LIN {X 0,Y 580.158,Z 386.279,A -85,B 0,C 180,E1 -1986.958,E2 -1986.958} C_VEL
LIN {X 0,Y 580.242,Z 378.359,A -85,B 0,C 180,E1 -1988.007,E2 -1988.007} C_VEL
LIN {X 0,Y 580.308,Z 368.509,A -85,B 0,C 180,E1 -1989.058,E2 -1989.058} C_VEL
LIN {X 0,Y 580.415,Z 358.188,A -85,B 0,C 180,E1 -1989.936,E2 -1989.936} C_VEL
LIN {X 0,Y 580.533,Z 346.552,A -85,B 0,C 180,E1 -1990.727,E2 -1990.727} C_VEL
LIN {X 0,Y 580.614,Z 334.997,A -85,B 0,C 180,E1 -1991.344,E2 -1991.344} C_VEL
LIN {X 0,Y 580.632,Z 322.991,A -85,B 0,C 180,E1 -1991.83,E2 -1991.83} C_VEL
LIN {X 0,Y 580.756,Z 309.958,A -85,B 0,C 180,E1 -1992.204,E2 -1992.204} C_VEL
LIN {X 0,Y 580.802,Z 297.624,A -85,B 0,C 180,E1 -1992.425,E2 -1992.425} C_VEL
LIN {X 0,Y 580.926,Z 253.863,A -85,B 0,C 180,E1 -1992.966,E2 -1992.966} C_VEL
LIN {X 0,Y 580.276,Z 248.059,A -85,B 0,C 180,E1 -1993.053,E2 -1993.053} C_VEL
LIN {X 0,Y 574.724,Z 229.373,A -85,B 0,C 180,E1 -1993.416,E2 -1993.416} C_VEL
LIN {X 0,Y 574.032,Z 223.57,A -85,B 0,C 180,E1 -1993.505,E2 -1993.505} C_VEL
LIN {X 0,Y 573.952,Z 199.2,A -85,B 0,C 180,E1 -1993.814,E2 -1993.814} C_VEL
LIN {X 0,Y 573.397,Z 195.222,A -85,B 0,C 180,E1 -1993.896,E2 -1993.896} C_VEL
LIN {X 0,Y 573.541,Z 175.453,A -85,B 0,C 180,E1 -1996.722,E2 -1996.722} C_VEL
LIN {X 0,Y 573.812,Z 157.024,A -85,B 0,C 180,E1 -1999.422,E2 -1999.422} C_VEL
LIN {X 0,Y 574.091,Z 137.477,A -85,B 0,C 180,E1 -2002.303,E2 -2002.303} C_VEL
LIN {X 0,Y 573.843,Z 133.661,A -85,B 0,C 180,E1 -2002.883,E2 -2002.883} C_VEL
LIN {X 0,Y 573.232,Z 130.71,A -85,B 0,C 180,E1 -2003.377,E2 -2003.377} C_VEL
LIN {X 0,Y 573.247,Z 130.708,A -85,B 0,C 180,E1 -2005.411,E2 -2005.411} C_VEL
LIN {X 0,Y 573.226,Z 130.702,A -85,B 0,C 180,E1 -2008.565,E2 -2008.565} C_VEL
LIN {X 0,Y 573.222,Z 130.705,A -85,B 0,C 180,E1 -2010.994,E2 -2010.994} C_VEL
LIN {X 0,Y 573.268,Z 130.704,A -85,B 0,C 180,E1 -2013.524,E2 -2013.524} C_VEL
LIN {X 0,Y 573.197,Z 130.706,A -85,B 0,C 180,E1 -2016.053,E2 -2016.053} C_VEL
LIN {X 0,Y 573.242,Z 130.701,A -85,B 0,C 180,E1 -2018.702,E2 -2018.702} C_VEL
LIN {X 0,Y 573.218,Z 130.706,A -85,B 0,C 180,E1 -2021.591,E2 -2021.591} C_VEL
LIN {X 0,Y 573.229,Z 130.7,A -85,B 0,C 180,E1 -2024.334,E2 -2024.334} C_VEL
LIN {X 0,Y 573.242,Z 130.704,A -85,B 0,C 180,E1 -2027.358,E2 -2027.358} C_VEL
LIN {X 0,Y 573.241,Z 130.701,A -85,B 0,C 180,E1 -2030.392,E2 -2030.392} C_VEL
LIN {X 0,Y 573.256,Z 130.705,A -85,B 0,C 180,E1 -2033.077,E2 -2033.077} C_VEL
LIN {X 0,Y 573.26,Z 130.698,A -85,B 0,C 180,E1 -2035.67,E2 -2035.67} C_VEL
LIN {X 0,Y 573.243,Z 130.702,A -85,B 0,C 180,E1 -2038.184,E2 -2038.184} C_VEL
LIN {X 0,Y 573.263,Z 130.706,A -85,B 0,C 180,E1 -2040.633,E2 -2040.633} C_VEL
LIN {X 0,Y 573.239,Z 130.701,A -85,B 0,C 180,E1 -2043.507,E2 -2043.507} C_VEL
LIN {X 0,Y 573.231,Z 130.708,A -85,B 0,C 180,E1 -2046.134,E2 -2046.134} C_VEL
LIN {X 0,Y 573.288,Z 130.867,A -85,B 0,C 180,E1 -2046.773,E2 -2046.773} C_VEL
LIN {X 0,Y 574.099,Z 135.892,A -85,B 0,C 180,E1 -2047.507,E2 -2047.507} C_VEL
LIN {X 0,Y 573.843,Z 156.505,A -85,B 0,C 180,E1 -2050.382,E2 -2050.382} C_VEL
LIN {X 0,Y 573.897,Z 157.389,A -85,B 0,C 180,E1 -2050.451,E2 -2050.451} C_VEL
LIN {X 0,Y 575.176,Z 163.348,A -85,B 0,C 180,E1 -2050.573,E2 -2050.573} C_VEL
LIN {X 0,Y 574.754,Z 320.455,A -85,B 0,C 180,E1 -2052.605,E2 -2052.605} C_VEL
LIN {X 0,Y 574.634,Z 333.869,A -85,B 0,C 180,E1 -2052.88,E2 -2052.88} C_VEL
LIN {X 0,Y 574.472,Z 349.297,A -85,B 0,C 180,E1 -2053.337,E2 -2053.337} C_VEL
LIN {X 0,Y 574.303,Z 363.777,A -85,B 0,C 180,E1 -2053.926,E2 -2053.926} C_VEL
LIN {X 0,Y 574.121,Z 376.223,A -85,B 0,C 180,E1 -2054.558,E2 -2054.558} C_VEL
LIN {X 0,Y 573.959,Z 387.161,A -85,B 0,C 180,E1 -2055.222,E2 -2055.222} C_VEL
LIN {X 0,Y 573.735,Z 398.068,A -85,B 0,C 180,E1 -2055.999,E2 -2055.999} C_VEL
LIN {X 0,Y 573.576,Z 408.837,A -85,B 0,C 180,E1 -2056.898,E2 -2056.898} C_VEL
LIN {X 0,Y 573.4,Z 421.37,A -85,B 0,C 180,E1 -2058.152,E2 -2058.152} C_VEL
LIN {X 0,Y 573.312,Z 430.525,A -85,B 0,C 180,E1 -2059.257,E2 -2059.257} C_VEL
LIN {X 0,Y 573.195,Z 437.937,A -85,B 0,C 180,E1 -2060.293,E2 -2060.293} C_VEL
LIN {X 0,Y 573.113,Z 445.456,A -85,B 0,C 180,E1 -2061.537,E2 -2061.537} C_VEL
LIN {X 0,Y 573.05,Z 452.505,A -85,B 0,C 180,E1 -2062.955,E2 -2062.955} C_VEL
LIN {X 0,Y 573.055,Z 458.02,A -85,B 0,C 180,E1 -2064.369,E2 -2064.369} C_VEL
LIN {X 0,Y 573.008,Z 462.158,A -85,B 0,C 180,E1 -2065.779,E2 -2065.779} C_VEL
LIN {X 0,Y 572.954,Z 465.104,A -85,B 0,C 180,E1 -2067.187,E2 -2067.187} C_VEL
LIN {X 0,Y 572.943,Z 466.876,A -85,B 0,C 180,E1 -2068.593,E2 -2068.593} C_VEL
LIN {X 0,Y 572.936,Z 467.496,A -85,B 0,C 180,E1 -2069.999,E2 -2069.999} C_VEL
LIN {X 0,Y 572.945,Z 466.961,A -85,B 0,C 180,E1 -2071.405,E2 -2071.405} C_VEL
LIN {X 0,Y 572.956,Z 465.263,A -85,B 0,C 180,E1 -2072.811,E2 -2072.811} C_VEL
LIN {X 0,Y 573.008,Z 462.383,A -85,B 0,C 180,E1 -2074.219,E2 -2074.219} C_VEL
LIN {X 0,Y 573.054,Z 458.318,A -85,B 0,C 180,E1 -2075.63,E2 -2075.63} C_VEL
LIN {X 0,Y 573.048,Z 452.921,A -85,B 0,C 180,E1 -2077.044,E2 -2077.044} C_VEL
LIN {X 0,Y 573.102,Z 445.973,A -85,B 0,C 180,E1 -2078.461,E2 -2078.461} C_VEL
LIN {X 0,Y 573.188,Z 438.539,A -85,B 0,C 180,E1 -2079.705,E2 -2079.705} C_VEL
LIN {X 0,Y 573.286,Z 430.107,A -85,B 0,C 180,E1 -2080.889,E2 -2080.889} C_VEL
LIN {X 0,Y 573.404,Z 420.579,A -85,B 0,C 180,E1 -2082.025,E2 -2082.025} C_VEL
LIN {X 0,Y 573.6,Z 408.856,A -85,B 0,C 180,E1 -2083.19,E2 -2083.19} C_VEL
LIN {X 0,Y 573.743,Z 398.086,A -85,B 0,C 180,E1 -2084.09,E2 -2084.09} C_VEL
LIN {X 0,Y 573.978,Z 386.69,A -85,B 0,C 180,E1 -2084.899,E2 -2084.899} C_VEL
LIN {X 0,Y 574.141,Z 374.636,A -85,B 0,C 180,E1 -2085.622,E2 -2085.622} C_VEL
LIN {X 0,Y 574.335,Z 359.788,A -85,B 0,C 180,E1 -2086.345,E2 -2086.345} C_VEL
LIN {X 0,Y 574.5,Z 345.108,A -85,B 0,C 180,E1 -2086.889,E2 -2086.889} C_VEL
LIN {X 0,Y 574.637,Z 332.407,A -85,B 0,C 180,E1 -2087.244,E2 -2087.244} C_VEL
LIN {X 0,Y 574.742,Z 319.698,A -85,B 0,C 180,E1 -2087.498,E2 -2087.498} C_VEL
LIN {X 0,Y 575.098,Z 163.083,A -85,B 0,C 180,E1 -2089.523,E2 -2089.523} C_VEL
LIN {X 0,Y 573.846,Z 156.905,A -85,B 0,C 180,E1 -2089.652,E2 -2089.652} C_VEL
LIN {X 0,Y 574.089,Z 137.93,A -85,B 0,C 180,E1 -2092.302,E2 -2092.302} C_VEL
LIN {X 0,Y 573.891,Z 133.83,A -85,B 0,C 180,E1 -2092.88,E2 -2092.88} C_VEL
LIN {X 0,Y 573.25,Z 130.708,A -85,B 0,C 180,E1 -2093.374,E2 -2093.374} C_VEL
LIN {X 0,Y 573.263,Z 130.7,A -85,B 0,C 180,E1 -2096.189,E2 -2096.189} C_VEL
LIN {X 0,Y 573.236,Z 130.701,A -85,B 0,C 180,E1 -2098.563,E2 -2098.563} C_VEL
LIN {X 0,Y 573.232,Z 130.704,A -85,B 0,C 180,E1 -2100.992,E2 -2100.992} C_VEL
LIN {X 0,Y 573.285,Z 130.704,A -85,B 0,C 180,E1 -2103.527,E2 -2103.527} C_VEL
LIN {X 0,Y 573.256,Z 130.699,A -85,B 0,C 180,E1 -2106.047,E2 -2106.047} C_VEL
LIN {X 0,Y 573.243,Z 130.7,A -85,B 0,C 180,E1 -2108.7,E2 -2108.7} C_VEL
LIN {X 0,Y 573.248,Z 130.704,A -85,B 0,C 180,E1 -2111.595,E2 -2111.595} C_VEL
LIN {X 0,Y 573.233,Z 130.699,A -85,B 0,C 180,E1 -2114.332,E2 -2114.332} C_VEL
LIN {X 0,Y 573.233,Z 130.708,A -85,B 0,C 180,E1 -2117.357,E2 -2117.357} C_VEL
LIN {X 0,Y 573.241,Z 130.699,A -85,B 0,C 180,E1 -2120.392,E2 -2120.392} C_VEL
LIN {X 0,Y 573.249,Z 130.706,A -85,B 0,C 180,E1 -2123.077,E2 -2123.077} C_VEL
LIN {X 0,Y 573.267,Z 130.697,A -85,B 0,C 180,E1 -2125.671,E2 -2125.671} C_VEL
LIN {X 0,Y 573.241,Z 130.699,A -85,B 0,C 180,E1 -2128.184,E2 -2128.184} C_VEL
LIN {X 0,Y 573.261,Z 130.697,A -85,B 0,C 180,E1 -2130.634,E2 -2130.634} C_VEL
LIN {X 0,Y 573.242,Z 130.709,A -85,B 0,C 180,E1 -2133.024,E2 -2133.024} C_VEL
LIN {X 0,Y 573.266,Z 130.699,A -85,B 0,C 180,E1 -2135.366,E2 -2135.366} C_VEL
LIN {X 0,Y 573.222,Z 130.703,A -85,B 0,C 180,E1 -2138.419,E2 -2138.419} C_VEL
LIN {X 0,Y 573.27,Z 130.7,A -85,B 0,C 180,E1 -2140.727,E2 -2140.727} C_VEL
LIN {X 0,Y 573.25,Z 130.699,A -85,B 0,C 180,E1 -2143.622,E2 -2143.622} C_VEL
LIN {X 0,Y 573.23,Z 130.704,A -85,B 0,C 180,E1 -2146.529,E2 -2146.529} C_VEL
LIN {X 0,Y 573.273,Z 130.702,A -85,B 0,C 180,E1 -2148.734,E2 -2148.734} C_VEL
LIN {X 0,Y 573.281,Z 130.694,A -85,B 0,C 180,E1 -2151.54,E2 -2151.54} C_VEL
LIN {X 0,Y 573.285,Z 130.694,A -85,B 0,C 180,E1 -2154.372,E2 -2154.372} C_VEL
LIN {X 0,Y 573.305,Z 130.694,A -85,B 0,C 180,E1 -2157.189,E2 -2157.189} C_VEL
LIN {X 0,Y 573.307,Z 130.689,A -85,B 0,C 180,E1 -2160,E2 -2160} C_VEL
LIN {X 0,Y 573.304,Z 130.699,A -85,B 0,C 180,E1 -2162.811,E2 -2162.811} C_VEL
LIN {X 0,Y 573.284,Z 130.692,A -85,B 0,C 180,E1 -2165.628,E2 -2165.628} C_VEL
LIN {X 0,Y 573.297,Z 130.698,A -85,B 0,C 180,E1 -2168.459,E2 -2168.459} C_VEL
LIN {X 0,Y 573.288,Z 130.692,A -85,B 0,C 180,E1 -2171.312,E2 -2171.312} C_VEL
LIN {X 0,Y 573.27,Z 130.702,A -85,B 0,C 180,E1 -2174.425,E2 -2174.425} C_VEL
LIN {X 0,Y 573.25,Z 130.698,A -85,B 0,C 180,E1 -2177.112,E2 -2177.112} C_VEL
LIN {X 0,Y 573.248,Z 130.7,A -85,B 0,C 180,E1 -2180.077,E2 -2180.077} C_VEL
LIN {X 0,Y 573.262,Z 130.696,A -85,B 0,C 180,E1 -2183.154,E2 -2183.154} C_VEL
LIN {X 0,Y 573.243,Z 130.697,A -85,B 0,C 180,E1 -2185.411,E2 -2185.411} C_VEL
LIN {X 0,Y 573.255,Z 130.703,A -85,B 0,C 180,E1 -2188.032,E2 -2188.032} C_VEL
LIN {X 0,Y 573.229,Z 130.702,A -85,B 0,C 180,E1 -2190.885,E2 -2190.885} C_VEL
LIN {X 0,Y 573.252,Z 130.698,A -85,B 0,C 180,E1 -2193.525,E2 -2193.525} C_VEL
LIN {X 0,Y 573.252,Z 130.705,A -85,B 0,C 180,E1 -2196.049,E2 -2196.049} C_VEL
LIN {X 0,Y 573.236,Z 130.699,A -85,B 0,C 180,E1 -2198.702,E2 -2198.702} C_VEL
LIN {X 0,Y 573.245,Z 130.697,A -85,B 0,C 180,E1 -2201.597,E2 -2201.597} C_VEL
LIN {X 0,Y 573.227,Z 130.707,A -85,B 0,C 180,E1 -2204.334,E2 -2204.334} C_VEL
LIN {X 0,Y 573.235,Z 130.701,A -85,B 0,C 180,E1 -2207.359,E2 -2207.359} C_VEL
LIN {X 0,Y 573.24,Z 130.703,A -85,B 0,C 180,E1 -2210.394,E2 -2210.394} C_VEL
LIN {X 0,Y 573.249,Z 130.698,A -85,B 0,C 180,E1 -2213.079,E2 -2213.079} C_VEL
LIN {X 0,Y 573.262,Z 130.701,A -85,B 0,C 180,E1 -2215.672,E2 -2215.672} C_VEL
LIN {X 0,Y 573.235,Z 130.707,A -85,B 0,C 180,E1 -2218.186,E2 -2218.186} C_VEL
LIN {X 0,Y 573.272,Z 130.848,A -85,B 0,C 180,E1 -2221.126,E2 -2221.126} C_VEL
LIN {X 0,Y 575.621,Z 138.924,A -85,B 0,C 180,E1 -2221.93,E2 -2221.93} C_VEL
LIN {X 0,Y 575.388,Z 166.625,A -85,B 0,C 180,E1 -2224.207,E2 -2224.207} C_VEL
LIN {X 0,Y 574.969,Z 203.279,A -85,B 0,C 180,E1 -2227.166,E2 -2227.166} C_VEL
LIN {X 0,Y 574.482,Z 240.019,A -85,B 0,C 180,E1 -2230.117,E2 -2230.117} C_VEL
LIN {X 0,Y 574.453,Z 243.087,A -85,B 0,C 180,E1 -2230.361,E2 -2230.361} C_VEL
LIN {X 0,Y 575.213,Z 250.056,A -85,B 0,C 180,E1 -2230.487,E2 -2230.487} C_VEL
LIN {X 0,Y 574.75,Z 412.28,A -85,B 0,C 180,E1 -2232.584,E2 -2232.584} C_VEL
LIN {X 0,Y 574.612,Z 427.743,A -85,B 0,C 180,E1 -2232.931,E2 -2232.931} C_VEL
LIN {X 0,Y 574.435,Z 443.067,A -85,B 0,C 180,E1 -2233.429,E2 -2233.429} C_VEL
LIN {X 0,Y 574.264,Z 456.795,A -85,B 0,C 180,E1 -2234.018,E2 -2234.018} C_VEL
LIN {X 0,Y 574.035,Z 470.264,A -85,B 0,C 180,E1 -2234.739,E2 -2234.739} C_VEL
LIN {X 0,Y 573.858,Z 483.833,A -85,B 0,C 180,E1 -2235.632,E2 -2235.632} C_VEL
LIN {X 0,Y 573.634,Z 496.362,A -85,B 0,C 180,E1 -2236.63,E2 -2236.63} C_VEL
LIN {X 0,Y 573.476,Z 506.758,A -85,B 0,C 180,E1 -2237.617,E2 -2237.617} C_VEL
LIN {X 0,Y 573.284,Z 516.777,A -85,B 0,C 180,E1 -2238.735,E2 -2238.735} C_VEL
LIN {X 0,Y 573.242,Z 525.865,A -85,B 0,C 180,E1 -2239.939,E2 -2239.939} C_VEL
LIN {X 0,Y 573.132,Z 533.74,A -85,B 0,C 180,E1 -2241.184,E2 -2241.184} C_VEL
LIN {X 0,Y 573.074,Z 541.095,A -85,B 0,C 180,E1 -2242.603,E2 -2242.603} C_VEL
LIN {X 0,Y 573.042,Z 546.926,A -85,B 0,C 180,E1 -2244.017,E2 -2244.017} C_VEL
LIN {X 0,Y 572.951,Z 550.388,A -85,B 0,C 180,E1 -2245.075,E2 -2245.075} C_VEL
LIN {X 0,Y 573.004,Z 553.891,A -85,B 0,C 180,E1 -2246.485,E2 -2246.485} C_VEL
LIN {X 0,Y 572.938,Z 556.193,A -85,B 0,C 180,E1 -2247.892,E2 -2247.892} C_VEL
LIN {X 0,Y 572.938,Z 557.349,A -85,B 0,C 180,E1 -2249.298,E2 -2249.298} C_VEL
LIN {X 0,Y 572.938,Z 557.348,A -85,B 0,C 180,E1 -2250.704,E2 -2250.704} C_VEL
LIN {X 0,Y 572.938,Z 556.189,A -85,B 0,C 180,E1 -2252.11,E2 -2252.11} C_VEL
LIN {X 0,Y 573.004,Z 553.885,A -85,B 0,C 180,E1 -2253.517,E2 -2253.517} C_VEL
LIN {X 0,Y 572.951,Z 550.383,A -85,B 0,C 180,E1 -2254.927,E2 -2254.927} C_VEL
LIN {X 0,Y 573.014,Z 545.605,A -85,B 0,C 180,E1 -2256.338,E2 -2256.338} C_VEL
LIN {X 0,Y 573.094,Z 539.418,A -85,B 0,C 180,E1 -2257.753,E2 -2257.753} C_VEL
LIN {X 0,Y 573.136,Z 531.643,A -85,B 0,C 180,E1 -2259.174,E2 -2259.174} C_VEL
LIN {X 0,Y 573.271,Z 523.363,A -85,B 0,C 180,E1 -2260.419,E2 -2260.419} C_VEL
LIN {X 0,Y 573.387,Z 513.384,A -85,B 0,C 180,E1 -2261.669,E2 -2261.669} C_VEL
LIN {X 0,Y 573.568,Z 503.179,A -85,B 0,C 180,E1 -2262.742,E2 -2262.742} C_VEL
LIN {X 0,Y 573.742,Z 491.009,A -85,B 0,C 180,E1 -2263.82,E2 -2263.82} C_VEL
LIN {X 0,Y 573.964,Z 477.893,A -85,B 0,C 180,E1 -2264.782,E2 -2264.782} C_VEL
LIN {X 0,Y 574.145,Z 465.499,A -85,B 0,C 180,E1 -2265.532,E2 -2265.532} C_VEL
LIN {X 0,Y 574.339,Z 450.811,A -85,B 0,C 180,E1 -2266.256,E2 -2266.256} C_VEL
LIN {X 0,Y 574.528,Z 436.592,A -85,B 0,C 180,E1 -2266.799,E2 -2266.799} C_VEL
LIN {X 0,Y 574.693,Z 421.863,A -85,B 0,C 180,E1 -2267.215,E2 -2267.215} C_VEL
LIN {X 0,Y 574.732,Z 407.195,A -85,B 0,C 180,E1 -2267.495,E2 -2267.495} C_VEL
LIN {X 0,Y 575.125,Z 247.826,A -85,B 0,C 180,E1 -2269.545,E2 -2269.545} C_VEL
LIN {X 0,Y 574.453,Z 243.095,A -85,B 0,C 180,E1 -2269.638,E2 -2269.638} C_VEL
LIN {X 0,Y 574.913,Z 206.745,A -85,B 0,C 180,E1 -2272.554,E2 -2272.554} C_VEL
LIN {X 0,Y 575.267,Z 171.131,A -85,B 0,C 180,E1 -2275.412,E2 -2275.412} C_VEL
LIN {X 0,Y 575.517,Z 141.849,A -85,B 0,C 180,E1 -2277.792,E2 -2277.792} C_VEL
LIN {X 0,Y 575.483,Z 138.561,A -85,B 0,C 180,E1 -2278.065,E2 -2278.065} C_VEL
LIN {X 0,Y 573.254,Z 130.703,A -85,B 0,C 180,E1 -2278.865,E2 -2278.865} C_VEL
LIN {X 0,Y 573.238,Z 130.709,A -85,B 0,C 180,E1 -2281.816,E2 -2281.816} C_VEL
LIN {X 0,Y 573.262,Z 130.702,A -85,B 0,C 180,E1 -2284.33,E2 -2284.33} C_VEL
LIN {X 0,Y 573.235,Z 130.704,A -85,B 0,C 180,E1 -2287.164,E2 -2287.164} C_VEL
LIN {X 0,Y 573.231,Z 130.71,A -85,B 0,C 180,E1 -2289.609,E2 -2289.609} C_VEL
LIN {X 0,Y 573.213,Z 130.704,A -85,B 0,C 180,E1 -2292.639,E2 -2292.639} C_VEL
LIN {X 0,Y 573.215,Z 130.709,A -85,B 0,C 180,E1 -2295.665,E2 -2295.665} C_VEL
LIN {X 0,Y 573.182,Z 130.709,A -85,B 0,C 180,E1 -2298.539,E2 -2298.539} C_VEL
LIN {X 0,Y 573.216,Z 130.711,A -85,B 0,C 180,E1 -2301.296,E2 -2301.296} C_VEL
LIN {X 0,Y 573.179,Z 130.709,A -85,B 0,C 180,E1 -2304.024,E2 -2304.024} C_VEL
LIN {X 0,Y 573.224,Z 130.707,A -85,B 0,C 180,E1 -2306.515,E2 -2306.515} C_VEL
LIN {X 0,Y 573.214,Z 130.709,A -85,B 0,C 180,E1 -2309.121,E2 -2309.121} C_VEL
LIN {X 0,Y 573.2,Z 130.708,A -85,B 0,C 180,E1 -2311.434,E2 -2311.434} C_VEL
LIN {X 0,Y 573.24,Z 130.704,A -85,B 0,C 180,E1 -2313.809,E2 -2313.809} C_VEL
LIN {X 0,Y 573.241,Z 130.752,A -85,B 0,C 180,E1 -2316.545,E2 -2316.545} C_VEL
LIN {X 0,Y 574.306,Z 136.752,A -85,B 0,C 180,E1 -2317.517,E2 -2317.517} C_VEL
LIN {X 0,Y 573.923,Z 156.686,A -85,B 0,C 180,E1 -2320.547,E2 -2320.547} C_VEL
LIN {X 0,Y 573.591,Z 174.992,A -85,B 0,C 180,E1 -2323.279,E2 -2323.279} C_VEL
LIN {X 0,Y 573.398,Z 193.795,A -85,B 0,C 180,E1 -2325.991,E2 -2325.991} C_VEL
LIN {X 0,Y 573.428,Z 195.663,A -85,B 0,C 180,E1 -2326.218,E2 -2326.218} C_VEL
LIN {X 0,Y 574.081,Z 201.024,A -85,B 0,C 180,E1 -2326.302,E2 -2326.302} C_VEL
LIN {X 0,Y 573.896,Z 303.446,A -85,B 0,C 180,E1 -2327.603,E2 -2327.603} C_VEL
LIN {X 0,Y 573.823,Z 315.958,A -85,B 0,C 180,E1 -2327.893,E2 -2327.893} C_VEL
LIN {X 0,Y 573.709,Z 327.744,A -85,B 0,C 180,E1 -2328.294,E2 -2328.294} C_VEL
LIN {X 0,Y 573.602,Z 339.246,A -85,B 0,C 180,E1 -2328.82,E2 -2328.82} C_VEL
LIN {X 0,Y 573.457,Z 350.757,A -85,B 0,C 180,E1 -2329.496,E2 -2329.496} C_VEL
LIN {X 0,Y 573.333,Z 361.499,A -85,B 0,C 180,E1 -2330.297,E2 -2330.297} C_VEL
LIN {X 0,Y 573.242,Z 371.164,A -85,B 0,C 180,E1 -2331.185,E2 -2331.185} C_VEL
LIN {X 0,Y 573.161,Z 379.087,A -85,B 0,C 180,E1 -2332.071,E2 -2332.071} C_VEL
LIN {X 0,Y 573.093,Z 387.023,A -85,B 0,C 180,E1 -2333.163,E2 -2333.163} C_VEL
LIN {X 0,Y 573.071,Z 393.948,A -85,B 0,C 180,E1 -2334.37,E2 -2334.37} C_VEL
LIN {X 0,Y 573.029,Z 398.691,A -85,B 0,C 180,E1 -2335.428,E2 -2335.428} C_VEL
LIN {X 0,Y 573.023,Z 402.324,A -85,B 0,C 180,E1 -2336.484,E2 -2336.484} C_VEL
LIN {X 0,Y 572.959,Z 404.2,A -85,B 0,C 180,E1 -2337.188,E2 -2337.188} C_VEL
LIN {X 0,Y 572.938,Z 405.625,A -85,B 0,C 180,E1 -2337.891,E2 -2337.891} C_VEL
LIN {X 0,Y 572.942,Z 407.256,A -85,B 0,C 180,E1 -2339.297,E2 -2339.297} C_VEL
LIN {X 0,Y 572.938,Z 407.496,A -85,B 0,C 180,E1 -2340,E2 -2340} C_VEL
LIN {X 0,Y 572.941,Z 407.315,A -85,B 0,C 180,E1 -2340.703,E2 -2340.703} C_VEL
LIN {X 0,Y 572.937,Z 405.771,A -85,B 0,C 180,E1 -2342.109,E2 -2342.109} C_VEL
LIN {X 0,Y 572.96,Z 404.411,A -85,B 0,C 180,E1 -2342.812,E2 -2342.812} C_VEL
LIN {X 0,Y 573.015,Z 401.531,A -85,B 0,C 180,E1 -2343.868,E2 -2343.868} C_VEL
LIN {X 0,Y 572.963,Z 397.63,A -85,B 0,C 180,E1 -2344.926,E2 -2344.926} C_VEL
LIN {X 0,Y 573.076,Z 392.601,A -85,B 0,C 180,E1 -2345.984,E2 -2345.984} C_VEL
LIN {X 0,Y 573.084,Z 386.275,A -85,B 0,C 180,E1 -2347.044,E2 -2347.044} C_VEL
LIN {X 0,Y 573.175,Z 378.354,A -85,B 0,C 180,E1 -2348.106,E2 -2348.106} C_VEL
LIN {X 0,Y 573.287,Z 368.502,A -85,B 0,C 180,E1 -2349.17,E2 -2349.17} C_VEL
LIN {X 0,Y 573.418,Z 358.182,A -85,B 0,C 180,E1 -2350.059,E2 -2350.059} C_VEL
LIN {X 0,Y 573.549,Z 346.568,A -85,B 0,C 180,E1 -2350.858,E2 -2350.858} C_VEL
LIN {X 0,Y 573.644,Z 334.987,A -85,B 0,C 180,E1 -2351.483,E2 -2351.483} C_VEL
LIN {X 0,Y 573.694,Z 322.973,A -85,B 0,C 180,E1 -2351.975,E2 -2351.975} C_VEL
LIN {X 0,Y 573.832,Z 309.933,A -85,B 0,C 180,E1 -2352.354,E2 -2352.354} C_VEL
LIN {X 0,Y 573.894,Z 297.583,A -85,B 0,C 180,E1 -2352.577,E2 -2352.577} C_VEL
LIN {X 0,Y 574.032,Z 223.57,A -85,B 0,C 180,E1 -2353.505,E2 -2353.505} C_VEL
LIN {X 0,Y 573.334,Z 219.693,A -85,B 0,C 180,E1 -2353.571,E2 -2353.571} C_VEL
LIN {X 0,Y 567.78,Z 207.719,A -85,B 0,C 180,E1 -2353.858,E2 -2353.858} C_VEL
LIN {X 0,Y 567.169,Z 203.842,A -85,B 0,C 180,E1 -2353.923,E2 -2353.923} C_VEL
LIN {X 0,Y 566.752,Z 197.824,A -85,B 0,C 180,E1 -2354.011,E2 -2354.011} C_VEL
LIN {X 0,Y 566.395,Z 195.238,A -85,B 0,C 180,E1 -2354.071,E2 -2354.071} C_VEL
LIN {X 0,Y 566.615,Z 174.482,A -85,B 0,C 180,E1 -2357.108,E2 -2357.108} C_VEL
LIN {X 0,Y 566.898,Z 155.433,A -85,B 0,C 180,E1 -2359.933,E2 -2359.933} C_VEL
LIN {X 0,Y 567.204,Z 137.62,A -85,B 0,C 180,E1 -2362.589,E2 -2362.589} C_VEL
LIN {X 0,Y 566.196,Z 131.587,A -85,B 0,C 180,E1 -2363.549,E2 -2363.549} C_VEL
LIN {X 0,Y 566.202,Z 131.585,A -85,B 0,C 180,E1 -2365.75,E2 -2365.75} C_VEL
LIN {X 0,Y 566.189,Z 131.58,A -85,B 0,C 180,E1 -2368.198,E2 -2368.198} C_VEL
LIN {X 0,Y 566.189,Z 131.583,A -85,B 0,C 180,E1 -2371.075,E2 -2371.075} C_VEL
LIN {X 0,Y 566.216,Z 131.579,A -85,B 0,C 180,E1 -2373.734,E2 -2373.734} C_VEL
LIN {X 0,Y 566.186,Z 131.579,A -85,B 0,C 180,E1 -2376.571,E2 -2376.571} C_VEL
LIN {X 0,Y 566.219,Z 131.575,A -85,B 0,C 180,E1 -2379.685,E2 -2379.685} C_VEL
LIN {X 0,Y 566.197,Z 131.583,A -85,B 0,C 180,E1 -2382.916,E2 -2382.916} C_VEL
LIN {X 0,Y 566.199,Z 131.577,A -85,B 0,C 180,E1 -2386.049,E2 -2386.049} C_VEL
LIN {X 0,Y 566.208,Z 131.58,A -85,B 0,C 180,E1 -2389.214,E2 -2389.214} C_VEL
LIN {X 0,Y 566.187,Z 131.58,A -85,B 0,C 180,E1 -2391.636,E2 -2391.636} C_VEL
LIN {X 0,Y 566.166,Z 131.584,A -85,B 0,C 180,E1 -2394.307,E2 -2394.307} C_VEL
LIN {X 0,Y 566.205,Z 131.584,A -85,B 0,C 180,E1 -2396.896,E2 -2396.896} C_VEL
LIN {X 0,Y 566.177,Z 131.581,A -85,B 0,C 180,E1 -2399.406,E2 -2399.406} C_VEL
LIN {X 0,Y 566.199,Z 131.578,A -85,B 0,C 180,E1 -2401.856,E2 -2401.856} C_VEL
LIN {X 0,Y 566.214,Z 131.581,A -85,B 0,C 180,E1 -2404.25,E2 -2404.25} C_VEL
LIN {X 0,Y 566.21,Z 131.7,A -85,B 0,C 180,E1 -2406.572,E2 -2406.572} C_VEL
LIN {X 0,Y 567.225,Z 137.371,A -85,B 0,C 180,E1 -2407.412,E2 -2407.412} C_VEL
LIN {X 0,Y 566.947,Z 156.955,A -85,B 0,C 180,E1 -2410.169,E2 -2410.169} C_VEL
LIN {X 0,Y 567.679,Z 160.632,A -85,B 0,C 180,E1 -2410.269,E2 -2410.269} C_VEL
LIN {X 0,Y 568.479,Z 165.015,A -85,B 0,C 180,E1 -2410.356,E2 -2410.356} C_VEL
LIN {X 0,Y 567.996,Z 320.772,A -85,B 0,C 180,E1 -2412.397,E2 -2412.397} C_VEL
LIN {X 0,Y 567.871,Z 333.383,A -85,B 0,C 180,E1 -2412.659,E2 -2412.659} C_VEL
LIN {X 0,Y 567.684,Z 347.978,A -85,B 0,C 180,E1 -2413.085,E2 -2413.085} C_VEL
LIN {X 0,Y 567.474,Z 363.767,A -85,B 0,C 180,E1 -2413.727,E2 -2413.727} C_VEL
LIN {X 0,Y 567.244,Z 376.215,A -85,B 0,C 180,E1 -2414.366,E2 -2414.366} C_VEL
LIN {X 0,Y 567.039,Z 387.577,A -85,B 0,C 180,E1 -2415.066,E2 -2415.066} C_VEL
LIN {X 0,Y 566.797,Z 399.243,A -85,B 0,C 180,E1 -2415.915,E2 -2415.915} C_VEL
LIN {X 0,Y 566.573,Z 410.825,A -85,B 0,C 180,E1 -2416.915,E2 -2416.915} C_VEL
LIN {X 0,Y 566.402,Z 421.364,A -85,B 0,C 180,E1 -2418.004,E2 -2418.004} C_VEL
LIN {X 0,Y 566.264,Z 429.936,A -85,B 0,C 180,E1 -2419.043,E2 -2419.043} C_VEL
LIN {X 0,Y 566.13,Z 437.93,A -85,B 0,C 180,E1 -2420.171,E2 -2420.171} C_VEL
LIN {X 0,Y 566.064,Z 445.451,A -85,B 0,C 180,E1 -2421.431,E2 -2421.431} C_VEL
LIN {X 0,Y 565.975,Z 452.51,A -85,B 0,C 180,E1 -2422.866,E2 -2422.866} C_VEL
LIN {X 0,Y 565.982,Z 458.018,A -85,B 0,C 180,E1 -2424.298,E2 -2424.298} C_VEL
LIN {X 0,Y 565.913,Z 462.153,A -85,B 0,C 180,E1 -2425.726,E2 -2425.726} C_VEL
LIN {X 0,Y 565.872,Z 465.097,A -85,B 0,C 180,E1 -2427.152,E2 -2427.152} C_VEL
LIN {X 0,Y 565.842,Z 466.87,A -85,B 0,C 180,E1 -2428.576,E2 -2428.576} C_VEL
LIN {X 0,Y 565.837,Z 467.496,A -85,B 0,C 180,E1 -2429.999,E2 -2429.999} C_VEL
LIN {X 0,Y 565.844,Z 466.96,A -85,B 0,C 180,E1 -2431.422,E2 -2431.422} C_VEL
LIN {X 0,Y 565.874,Z 465.254,A -85,B 0,C 180,E1 -2432.847,E2 -2432.847} C_VEL
LIN {X 0,Y 565.913,Z 462.375,A -85,B 0,C 180,E1 -2434.272,E2 -2434.272} C_VEL
LIN {X 0,Y 565.982,Z 458.308,A -85,B 0,C 180,E1 -2435.7,E2 -2435.7} C_VEL
LIN {X 0,Y 565.973,Z 452.918,A -85,B 0,C 180,E1 -2437.132,E2 -2437.132} C_VEL
LIN {X 0,Y 566.058,Z 445.962,A -85,B 0,C 180,E1 -2438.567,E2 -2438.567} C_VEL
LIN {X 0,Y 566.124,Z 438.524,A -85,B 0,C 180,E1 -2439.827,E2 -2439.827} C_VEL
LIN {X 0,Y 566.252,Z 430.621,A -85,B 0,C 180,E1 -2440.956,E2 -2440.956} C_VEL
LIN {X 0,Y 566.413,Z 420.578,A -85,B 0,C 180,E1 -2442.176,E2 -2442.176} C_VEL
LIN {X 0,Y 566.611,Z 408.835,A -85,B 0,C 180,E1 -2443.356,E2 -2443.356} C_VEL
LIN {X 0,Y 566.802,Z 398.065,A -85,B 0,C 180,E1 -2444.266,E2 -2444.266} C_VEL
LIN {X 0,Y 567.042,Z 387.744,A -85,B 0,C 180,E1 -2445.013,E2 -2445.013} C_VEL
LIN {X 0,Y 567.193,Z 377.813,A -85,B 0,C 180,E1 -2445.633,E2 -2445.633} C_VEL
LIN {X 0,Y 567.416,Z 365.659,A -85,B 0,C 180,E1 -2446.273,E2 -2446.273} C_VEL
LIN {X 0,Y 567.57,Z 354.02,A -85,B 0,C 180,E1 -2446.777,E2 -2446.777} C_VEL
LIN {X 0,Y 567.787,Z 339.987,A -85,B 0,C 180,E1 -2447.257,E2 -2447.257} C_VEL
LIN {X 0,Y 567.941,Z 324.406,A -85,B 0,C 180,E1 -2447.634,E2 -2447.634} C_VEL
LIN {X 0,Y 568.048,Z 300.042,A -85,B 0,C 180,E1 -2447.982,E2 -2447.982} C_VEL
LIN {X 0,Y 568.432,Z 164.207,A -85,B 0,C 180,E1 -2449.746,E2 -2449.746} C_VEL
LIN {X 0,Y 566.934,Z 157.091,A -85,B 0,C 180,E1 -2449.901,E2 -2449.901} C_VEL
LIN {X 0,Y 567.218,Z 139.41,A -85,B 0,C 180,E1 -2452.395,E2 -2452.395} C_VEL
LIN {X 0,Y 566.987,Z 135.364,A -85,B 0,C 180,E1 -2452.972,E2 -2452.972} C_VEL
LIN {X 0,Y 566.213,Z 131.585,A -85,B 0,C 180,E1 -2453.547,E2 -2453.547} C_VEL
LIN {X 0,Y 566.213,Z 131.584,A -85,B 0,C 180,E1 -2455.748,E2 -2455.748} C_VEL
LIN {X 0,Y 566.199,Z 131.579,A -85,B 0,C 180,E1 -2458.201,E2 -2458.201} C_VEL
LIN {X 0,Y 566.196,Z 131.582,A -85,B 0,C 180,E1 -2461.077,E2 -2461.077} C_VEL
LIN {X 0,Y 566.225,Z 131.579,A -85,B 0,C 180,E1 -2463.736,E2 -2463.736} C_VEL
LIN {X 0,Y 566.212,Z 131.575,A -85,B 0,C 180,E1 -2466.568,E2 -2466.568} C_VEL
LIN {X 0,Y 566.207,Z 131.576,A -85,B 0,C 180,E1 -2469.685,E2 -2469.685} C_VEL
LIN {X 0,Y 566.208,Z 131.576,A -85,B 0,C 180,E1 -2472.086,E2 -2472.086} C_VEL
LIN {X 0,Y 566.166,Z 131.585,A -85,B 0,C 180,E1 -2475.035,E2 -2475.035} C_VEL
LIN {X 0,Y 566.21,Z 131.575,A -85,B 0,C 180,E1 -2478.135,E2 -2478.135} C_VEL
LIN {X 0,Y 566.215,Z 131.577,A -85,B 0,C 180,E1 -2480.726,E2 -2480.726} C_VEL
LIN {X 0,Y 566.21,Z 131.576,A -85,B 0,C 180,E1 -2483.782,E2 -2483.782} C_VEL
LIN {X 0,Y 566.204,Z 131.575,A -85,B 0,C 180,E1 -2486.265,E2 -2486.265} C_VEL
LIN {X 0,Y 566.195,Z 131.584,A -85,B 0,C 180,E1 -2488.92,E2 -2488.92} C_VEL
LIN {X 0,Y 566.188,Z 131.584,A -85,B 0,C 180,E1 -2491.046,E2 -2491.046} C_VEL
LIN {X 0,Y 566.208,Z 131.578,A -85,B 0,C 180,E1 -2493.458,E2 -2493.458} C_VEL
LIN {X 0,Y 566.191,Z 131.576,A -85,B 0,C 180,E1 -2495.819,E2 -2495.819} C_VEL
LIN {X 0,Y 566.207,Z 131.584,A -85,B 0,C 180,E1 -2498.902,E2 -2498.902} C_VEL
LIN {X 0,Y 566.203,Z 131.581,A -85,B 0,C 180,E1 -2501.172,E2 -2501.172} C_VEL
LIN {X 0,Y 566.212,Z 131.577,A -85,B 0,C 180,E1 -2503.412,E2 -2503.412} C_VEL
LIN {X 0,Y 566.192,Z 131.578,A -85,B 0,C 180,E1 -2506.359,E2 -2506.359} C_VEL
LIN {X 0,Y 566.265,Z 131.573,A -85,B 0,C 180,E1 -2508.654,E2 -2508.654} C_VEL
LIN {X 0,Y 566.225,Z 131.574,A -85,B 0,C 180,E1 -2511.434,E2 -2511.434} C_VEL
LIN {X 0,Y 566.252,Z 131.569,A -85,B 0,C 180,E1 -2514.302,E2 -2514.302} C_VEL
LIN {X 0,Y 566.268,Z 131.568,A -85,B 0,C 180,E1 -2517.866,E2 -2517.866} C_VEL
LIN {X 0,Y 566.3,Z 131.57,A -85,B 0,C 180,E1 -2520.711,E2 -2520.711} C_VEL
LIN {X 0,Y 566.269,Z 131.574,A -85,B 0,C 180,E1 -2522.845,E2 -2522.845} C_VEL
LIN {X 0,Y 566.251,Z 131.568,A -85,B 0,C 180,E1 -2525.698,E2 -2525.698} C_VEL
LIN {X 0,Y 566.239,Z 131.579,A -85,B 0,C 180,E1 -2528.565,E2 -2528.565} C_VEL
LIN {X 0,Y 566.24,Z 131.57,A -85,B 0,C 180,E1 -2531.454,E2 -2531.454} C_VEL
LIN {X 0,Y 566.223,Z 131.581,A -85,B 0,C 180,E1 -2534.507,E2 -2534.507} C_VEL
LIN {X 0,Y 566.194,Z 131.576,A -85,B 0,C 180,E1 -2537.332,E2 -2537.332} C_VEL
LIN {X 0,Y 566.21,Z 131.581,A -85,B 0,C 180,E1 -2540.337,E2 -2540.337} C_VEL
LIN {X 0,Y 566.22,Z 131.572,A -85,B 0,C 180,E1 -2543.402,E2 -2543.402} C_VEL
LIN {X 0,Y 566.203,Z 131.576,A -85,B 0,C 180,E1 -2545.749,E2 -2545.749} C_VEL
LIN {X 0,Y 566.198,Z 131.585,A -85,B 0,C 180,E1 -2548.204,E2 -2548.204} C_VEL
LIN {X 0,Y 566.19,Z 131.578,A -85,B 0,C 180,E1 -2551.079,E2 -2551.079} C_VEL
LIN {X 0,Y 566.202,Z 131.578,A -85,B 0,C 180,E1 -2553.735,E2 -2553.735} C_VEL
LIN {X 0,Y 566.208,Z 131.579,A -85,B 0,C 180,E1 -2556.569,E2 -2556.569} C_VEL
LIN {X 0,Y 566.2,Z 131.575,A -85,B 0,C 180,E1 -2559.686,E2 -2559.686} C_VEL
LIN {X 0,Y 566.205,Z 131.581,A -85,B 0,C 180,E1 -2562.088,E2 -2562.088} C_VEL
LIN {X 0,Y 566.166,Z 131.581,A -85,B 0,C 180,E1 -2565.037,E2 -2565.037} C_VEL
LIN {X 0,Y 566.211,Z 131.584,A -85,B 0,C 180,E1 -2568.137,E2 -2568.137} C_VEL
LIN {X 0,Y 566.214,Z 131.575,A -85,B 0,C 180,E1 -2570.728,E2 -2570.728} C_VEL
LIN {X 0,Y 566.208,Z 131.581,A -85,B 0,C 180,E1 -2573.785,E2 -2573.785} C_VEL
LIN {X 0,Y 566.223,Z 131.574,A -85,B 0,C 180,E1 -2576.899,E2 -2576.899} C_VEL
LIN {X 0,Y 566.181,Z 131.584,A -85,B 0,C 180,E1 -2579.409,E2 -2579.409} C_VEL
LIN {X 0,Y 566.237,Z 131.676,A -85,B 0,C 180,E1 -2580.834,E2 -2580.834} C_VEL
LIN {X 0,Y 568.803,Z 140.456,A -85,B 0,C 180,E1 -2581.726,E2 -2581.726} C_VEL
LIN {X 0,Y 568.892,Z 151.97,A -85,B 0,C 180,E1 -2582.702,E2 -2582.702} C_VEL
LIN {X 0,Y 568.375,Z 184.986,A -85,B 0,C 180,E1 -2585.433,E2 -2585.433} C_VEL
LIN {X 0,Y 567.979,Z 217.542,A -85,B 0,C 180,E1 -2588.056,E2 -2588.056} C_VEL
LIN {X 0,Y 567.643,Z 243.149,A -85,B 0,C 180,E1 -2590.121,E2 -2590.121} C_VEL
LIN {X 0,Y 568.522,Z 250.001,A -85,B 0,C 180,E1 -2590.247,E2 -2590.247} C_VEL
LIN {X 0,Y 567.993,Z 412.233,A -85,B 0,C 180,E1 -2592.369,E2 -2592.369} C_VEL
LIN {X 0,Y 567.825,Z 427.741,A -85,B 0,C 180,E1 -2592.721,E2 -2592.721} C_VEL
LIN {X 0,Y 567.635,Z 443.064,A -85,B 0,C 180,E1 -2593.225,E2 -2593.225} C_VEL
LIN {X 0,Y 567.403,Z 456.799,A -85,B 0,C 180,E1 -2593.819,E2 -2593.819} C_VEL
LIN {X 0,Y 567.147,Z 470.266,A -85,B 0,C 180,E1 -2594.549,E2 -2594.549} C_VEL
LIN {X 0,Y 566.929,Z 482.536,A -85,B 0,C 180,E1 -2595.36,E2 -2595.36} C_VEL
LIN {X 0,Y 566.671,Z 495.303,A -85,B 0,C 180,E1 -2596.372,E2 -2596.372} C_VEL
LIN {X 0,Y 566.49,Z 506.758,A -85,B 0,C 180,E1 -2597.462,E2 -2597.462} C_VEL
LIN {X 0,Y 566.267,Z 517.318,A -85,B 0,C 180,E1 -2598.66,E2 -2598.66} C_VEL
LIN {X 0,Y 566.208,Z 525.864,A -85,B 0,C 180,E1 -2599.813,E2 -2599.813} C_VEL
LIN {X 0,Y 566.057,Z 533.741,A -85,B 0,C 180,E1 -2601.073,E2 -2601.073} C_VEL
LIN {X 0,Y 565.996,Z 541.095,A -85,B 0,C 180,E1 -2602.509,E2 -2602.509} C_VEL
LIN {X 0,Y 565.958,Z 546.926,A -85,B 0,C 180,E1 -2603.942,E2 -2603.942} C_VEL
LIN {X 0,Y 565.866,Z 550.388,A -85,B 0,C 180,E1 -2605.013,E2 -2605.013} C_VEL
LIN {X 0,Y 565.909,Z 553.891,A -85,B 0,C 180,E1 -2606.441,E2 -2606.441} C_VEL
LIN {X 0,Y 565.839,Z 556.192,A -85,B 0,C 180,E1 -2607.866,E2 -2607.866} C_VEL
LIN {X 0,Y 565.839,Z 557.349,A -85,B 0,C 180,E1 -2609.289,E2 -2609.289} C_VEL
LIN {X 0,Y 565.839,Z 557.348,A -85,B 0,C 180,E1 -2610.713,E2 -2610.713} C_VEL
LIN {X 0,Y 565.839,Z 556.188,A -85,B 0,C 180,E1 -2612.136,E2 -2612.136} C_VEL
LIN {X 0,Y 565.909,Z 553.885,A -85,B 0,C 180,E1 -2613.561,E2 -2613.561} C_VEL
LIN {X 0,Y 565.867,Z 550.383,A -85,B 0,C 180,E1 -2614.988,E2 -2614.988} C_VEL
LIN {X 0,Y 565.943,Z 545.605,A -85,B 0,C 180,E1 -2616.418,E2 -2616.418} C_VEL
LIN {X 0,Y 566.015,Z 539.418,A -85,B 0,C 180,E1 -2617.851,E2 -2617.851} C_VEL
LIN {X 0,Y 566.071,Z 531.641,A -85,B 0,C 180,E1 -2619.289,E2 -2619.289} C_VEL
LIN {X 0,Y 566.24,Z 523.362,A -85,B 0,C 180,E1 -2620.55,E2 -2620.55} C_VEL
LIN {X 0,Y 566.368,Z 513.385,A -85,B 0,C 180,E1 -2621.815,E2 -2621.815} C_VEL
LIN {X 0,Y 566.586,Z 503.178,A -85,B 0,C 180,E1 -2622.902,E2 -2622.902} C_VEL
LIN {X 0,Y 566.801,Z 491.009,A -85,B 0,C 180,E1 -2623.993,E2 -2623.993} C_VEL
LIN {X 0,Y 567.042,Z 478.326,A -85,B 0,C 180,E1 -2624.937,E2 -2624.937} C_VEL
LIN {X 0,Y 567.271,Z 465.495,A -85,B 0,C 180,E1 -2625.725,E2 -2625.725} C_VEL
LIN {X 0,Y 567.495,Z 450.808,A -85,B 0,C 180,E1 -2626.457,E2 -2626.457} C_VEL
LIN {X 0,Y 567.737,Z 436.591,A -85,B 0,C 180,E1 -2627.006,E2 -2627.006} C_VEL
LIN {X 0,Y 567.897,Z 421.633,A -85,B 0,C 180,E1 -2627.434,E2 -2627.434} C_VEL
LIN {X 0,Y 567.978,Z 406.956,A -85,B 0,C 180,E1 -2627.714,E2 -2627.714} C_VEL
LIN {X 0,Y 568.504,Z 249.661,A -85,B 0,C 180,E1 -2629.758,E2 -2629.758} C_VEL
LIN {X 0,Y 567.633,Z 243.053,A -85,B 0,C 180,E1 -2629.887,E2 -2629.887} C_VEL
LIN {X 0,Y 568.045,Z 209.813,A -85,B 0,C 180,E1 -2632.554,E2 -2632.554} C_VEL
LIN {X 0,Y 568.436,Z 177.26,A -85,B 0,C 180,E1 -2635.173,E2 -2635.173} C_VEL
LIN {X 0,Y 568.833,Z 145.38,A -85,B 0,C 180,E1 -2637.802,E2 -2637.802} C_VEL
LIN {X 0,Y 568.636,Z 140.071,A -85,B 0,C 180,E1 -2638.264,E2 -2638.264} C_VEL
LIN {X 0,Y 566.23,Z 131.578,A -85,B 0,C 180,E1 -2639.13,E2 -2639.13} C_VEL
LIN {X 0,Y 566.229,Z 131.581,A -85,B 0,C 180,E1 -2642.257,E2 -2642.257} C_VEL
LIN {X 0,Y 566.171,Z 131.583,A -85,B 0,C 180,E1 -2644.988,E2 -2644.988} C_VEL
LIN {X 0,Y 566.191,Z 131.585,A -85,B 0,C 180,E1 -2647.462,E2 -2647.462} C_VEL
LIN {X 0,Y 566.197,Z 131.58,A -85,B 0,C 180,E1 -2650.201,E2 -2650.201} C_VEL
LIN {X 0,Y 566.147,Z 131.588,A -85,B 0,C 180,E1 -2653.06,E2 -2653.06} C_VEL
LIN {X 0,Y 566.154,Z 131.584,A -85,B 0,C 180,E1 -2656.054,E2 -2656.054} C_VEL
LIN {X 0,Y 566.132,Z 131.59,A -85,B 0,C 180,E1 -2658.857,E2 -2658.857} C_VEL
LIN {X 0,Y 566.18,Z 131.585,A -85,B 0,C 180,E1 -2661.447,E2 -2661.447} C_VEL
LIN {X 0,Y 566.135,Z 131.587,A -85,B 0,C 180,E1 -2664.306,E2 -2664.306} C_VEL
LIN {X 0,Y 566.165,Z 131.591,A -85,B 0,C 180,E1 -2666.894,E2 -2666.894} C_VEL
LIN {X 0,Y 566.161,Z 131.585,A -85,B 0,C 180,E1 -2669.406,E2 -2669.406} C_VEL
LIN {X 0,Y 566.153,Z 131.585,A -85,B 0,C 180,E1 -2671.854,E2 -2671.854} C_VEL
LIN {X 0,Y 566.193,Z 131.586,A -85,B 0,C 180,E1 -2674.25,E2 -2674.25} C_VEL
LIN {X 0,Y 566.19,Z 131.752,A -85,B 0,C 180,E1 -2676.305,E2 -2676.305} C_VEL
LIN {X 0,Y 567.401,Z 137.312,A -85,B 0,C 180,E1 -2677.23,E2 -2677.23} C_VEL
LIN {X 0,Y 567.238,Z 150.909,A -85,B 0,C 180,E1 -2679.322,E2 -2679.322} C_VEL
LIN {X 0,Y 566.886,Z 169.609,A -85,B 0,C 180,E1 -2682.131,E2 -2682.131} C_VEL
LIN {X 0,Y 566.457,Z 189.121,A -85,B 0,C 180,E1 -2685.083,E2 -2685.083} C_VEL
LIN {X 0,Y 566.387,Z 195.464,A -85,B 0,C 180,E1 -2686.032,E2 -2686.032} C_VEL
LIN {X 0,Y 567.195,Z 201.139,A -85,B 0,C 180,E1 -2686.132,E2 -2686.132} C_VEL
LIN {X 0,Y 566.975,Z 303.475,A -85,B 0,C 180,E1 -2687.449,E2 -2687.449} C_VEL
LIN {X 0,Y 566.891,Z 316.74,A -85,B 0,C 180,E1 -2687.765,E2 -2687.765} C_VEL
LIN {X 0,Y 566.749,Z 328.887,A -85,B 0,C 180,E1 -2688.194,E2 -2688.194} C_VEL
LIN {X 0,Y 566.605,Z 341.151,A -85,B 0,C 180,E1 -2688.781,E2 -2688.781} C_VEL
LIN {X 0,Y 566.442,Z 352.055,A -85,B 0,C 180,E1 -2689.455,E2 -2689.455} C_VEL
LIN {X 0,Y 566.309,Z 362.573,A -85,B 0,C 180,E1 -2690.265,E2 -2690.265} C_VEL
LIN {X 0,Y 566.221,Z 371.17,A -85,B 0,C 180,E1 -2691.075,E2 -2691.075} C_VEL
LIN {X 0,Y 566.113,Z 379.091,A -85,B 0,C 180,E1 -2691.972,E2 -2691.972} C_VEL
LIN {X 0,Y 566.05,Z 385.656,A -85,B 0,C 180,E1 -2692.868,E2 -2692.868} C_VEL
LIN {X 0,Y 566.003,Z 392.126,A -85,B 0,C 180,E1 -2693.942,E2 -2693.942} C_VEL
LIN {X 0,Y 565.877,Z 397.265,A -85,B 0,C 180,E1 -2695.013,E2 -2695.013} C_VEL
LIN {X 0,Y 565.927,Z 401.254,A -85,B 0,C 180,E1 -2696.084,E2 -2696.084} C_VEL
LIN {X 0,Y 565.878,Z 404.202,A -85,B 0,C 180,E1 -2697.153,E2 -2697.153} C_VEL
LIN {X 0,Y 565.839,Z 405.625,A -85,B 0,C 180,E1 -2697.865,E2 -2697.865} C_VEL
LIN {X 0,Y 565.842,Z 407.256,A -85,B 0,C 180,E1 -2699.288,E2 -2699.288} C_VEL
LIN {X 0,Y 565.839,Z 407.496,A -85,B 0,C 180,E1 -2700,E2 -2700} C_VEL
LIN {X 0,Y 565.841,Z 407.316,A -85,B 0,C 180,E1 -2700.712,E2 -2700.712} C_VEL
LIN {X 0,Y 565.838,Z 405.77,A -85,B 0,C 180,E1 -2702.136,E2 -2702.136} C_VEL
LIN {X 0,Y 565.879,Z 404.409,A -85,B 0,C 180,E1 -2702.848,E2 -2702.848} C_VEL
LIN {X 0,Y 565.927,Z 401.529,A -85,B 0,C 180,E1 -2703.917,E2 -2703.917} C_VEL
LIN {X 0,Y 565.878,Z 397.628,A -85,B 0,C 180,E1 -2704.988,E2 -2704.988} C_VEL
LIN {X 0,Y 565.99,Z 392.599,A -85,B 0,C 180,E1 -2706.059,E2 -2706.059} C_VEL
LIN {X 0,Y 566.032,Z 386.271,A -85,B 0,C 180,E1 -2707.132,E2 -2707.132} C_VEL
LIN {X 0,Y 566.129,Z 378.348,A -85,B 0,C 180,E1 -2708.208,E2 -2708.208} C_VEL
LIN {X 0,Y 566.249,Z 368.496,A -85,B 0,C 180,E1 -2709.285,E2 -2709.285} C_VEL
LIN {X 0,Y 566.417,Z 358.172,A -85,B 0,C 180,E1 -2710.184,E2 -2710.184} C_VEL
LIN {X 0,Y 566.559,Z 346.81,A -85,B 0,C 180,E1 -2710.977,E2 -2710.977} C_VEL
LIN {X 0,Y 566.678,Z 334.976,A -85,B 0,C 180,E1 -2711.626,E2 -2711.626} C_VEL
LIN {X 0,Y 566.744,Z 322.955,A -85,B 0,C 180,E1 -2712.125,E2 -2712.125} C_VEL
LIN {X 0,Y 566.888,Z 309.909,A -85,B 0,C 180,E1 -2712.508,E2 -2712.508} C_VEL
LIN {X 0,Y 566.991,Z 297.541,A -85,B 0,C 180,E1 -2712.733,E2 -2712.733} C_VEL
LIN {X 0,Y 567.169,Z 203.842,A -85,B 0,C 180,E1 -2713.923,E2 -2713.923} C_VEL
LIN {X 0,Y 566.836,Z 200.194,A -85,B 0,C 180,E1 -2714.027,E2 -2714.027} C_VEL
LIN {X 0,Y 565.658,Z 196.194,A -85,B 0,C 180,E1 -2714.272,E2 -2714.272} C_VEL
LIN {X 0,Y 564.05,Z 192.825,A -85,B 0,C 180,E1 -2714.6,E2 -2714.6} C_VEL
LIN {X 0,Y 561.964,Z 189.409,A -85,B 0,C 180,E1 -2715.078,E2 -2715.078} C_VEL
LIN {X 0,Y 559.872,Z 185.11,A -85,B 0,C 180,E1 -2715.786,E2 -2715.786} C_VEL
LIN {X 0,Y 559.557,Z 182.779,A -85,B 0,C 180,E1 -2716.144,E2 -2716.144} C_VEL
LIN {X 0,Y 559.913,Z 163.274,A -85,B 0,C 180,E1 -2719.048,E2 -2719.048} C_VEL
LIN {X 0,Y 560.176,Z 145.68,A -85,B 0,C 180,E1 -2721.684,E2 -2721.684} C_VEL
LIN {X 0,Y 560.204,Z 137.73,A -85,B 0,C 180,E1 -2722.887,E2 -2722.887} C_VEL
LIN {X 0,Y 559.171,Z 132.462,A -85,B 0,C 180,E1 -2723.765,E2 -2723.765} C_VEL
LIN {X 0,Y 559.166,Z 132.457,A -85,B 0,C 180,E1 -2726.098,E2 -2726.098} C_VEL
LIN {X 0,Y 559.134,Z 132.458,A -85,B 0,C 180,E1 -2728.531,E2 -2728.531} C_VEL
LIN {X 0,Y 559.145,Z 132.463,A -85,B 0,C 180,E1 -2731.272,E2 -2731.272} C_VEL
LIN {X 0,Y 559.169,Z 132.454,A -85,B 0,C 180,E1 -2733.949,E2 -2733.949} C_VEL
LIN {X 0,Y 559.135,Z 132.464,A -85,B 0,C 180,E1 -2737.109,E2 -2737.109} C_VEL
LIN {X 0,Y 559.165,Z 132.452,A -85,B 0,C 180,E1 -2739.941,E2 -2739.941} C_VEL
LIN {X 0,Y 559.153,Z 132.458,A -85,B 0,C 180,E1 -2742.744,E2 -2742.744} C_VEL
LIN {X 0,Y 559.154,Z 132.455,A -85,B 0,C 180,E1 -2745.761,E2 -2745.761} C_VEL
LIN {X 0,Y 559.166,Z 132.454,A -85,B 0,C 180,E1 -2748.229,E2 -2748.229} C_VEL
LIN {X 0,Y 559.177,Z 132.458,A -85,B 0,C 180,E1 -2751.192,E2 -2751.192} C_VEL
LIN {X 0,Y 559.143,Z 132.457,A -85,B 0,C 180,E1 -2753.789,E2 -2753.789} C_VEL
LIN {X 0,Y 559.151,Z 132.46,A -85,B 0,C 180,E1 -2756.424,E2 -2756.424} C_VEL
LIN {X 0,Y 559.155,Z 132.461,A -85,B 0,C 180,E1 -2758.98,E2 -2758.98} C_VEL
LIN {X 0,Y 559.15,Z 132.456,A -85,B 0,C 180,E1 -2761.623,E2 -2761.623} C_VEL
LIN {X 0,Y 559.182,Z 132.454,A -85,B 0,C 180,E1 -2763.902,E2 -2763.902} C_VEL
LIN {X 0,Y 559.186,Z 132.611,A -85,B 0,C 180,E1 -2766.373,E2 -2766.373} C_VEL
LIN {X 0,Y 560.357,Z 138.9,A -85,B 0,C 180,E1 -2767.314,E2 -2767.314} C_VEL
LIN {X 0,Y 560.11,Z 157.496,A -85,B 0,C 180,E1 -2769.929,E2 -2769.929} C_VEL
LIN {X 0,Y 561.799,Z 165.492,A -85,B 0,C 180,E1 -2770.113,E2 -2770.113} C_VEL
LIN {X 0,Y 561.251,Z 321.178,A -85,B 0,C 180,E1 -2772.18,E2 -2772.18} C_VEL
LIN {X 0,Y 561.096,Z 336.074,A -85,B 0,C 180,E1 -2772.505,E2 -2772.505} C_VEL
LIN {X 0,Y 560.818,Z 351.726,A -85,B 0,C 180,E1 -2773.013,E2 -2773.013} C_VEL
LIN {X 0,Y 560.639,Z 363.756,A -85,B 0,C 180,E1 -2773.523,E2 -2773.523} C_VEL
LIN {X 0,Y 560.401,Z 374.605,A -85,B 0,C 180,E1 -2774.077,E2 -2774.077} C_VEL
LIN {X 0,Y 560.175,Z 386.356,A -85,B 0,C 180,E1 -2774.796,E2 -2774.796} C_VEL
LIN {X 0,Y 559.932,Z 396.874,A -85,B 0,C 180,E1 -2775.554,E2 -2775.554} C_VEL
LIN {X 0,Y 559.688,Z 406.77,A -85,B 0,C 180,E1 -2776.381,E2 -2776.381} C_VEL
LIN {X 0,Y 559.511,Z 416.248,A -85,B 0,C 180,E1 -2777.301,E2 -2777.301} C_VEL
LIN {X 0,Y 559.304,Z 426.02,A -85,B 0,C 180,E1 -2778.401,E2 -2778.401} C_VEL
LIN {X 0,Y 559.187,Z 435.577,A -85,B 0,C 180,E1 -2779.682,E2 -2779.682} C_VEL
LIN {X 0,Y 559.004,Z 443.447,A -85,B 0,C 180,E1 -2780.957,E2 -2780.957} C_VEL
LIN {X 0,Y 558.948,Z 449.164,A -85,B 0,C 180,E1 -2782.049,E2 -2782.049} C_VEL
LIN {X 0,Y 558.885,Z 453.986,A -85,B 0,C 180,E1 -2783.138,E2 -2783.138} C_VEL
LIN {X 0,Y 558.857,Z 459.139,A -85,B 0,C 180,E1 -2784.587,E2 -2784.587} C_VEL
LIN {X 0,Y 558.818,Z 463.821,A -85,B 0,C 180,E1 -2786.394,E2 -2786.394} C_VEL
LIN {X 0,Y 558.745,Z 466.13,A -85,B 0,C 180,E1 -2787.837,E2 -2787.837} C_VEL
LIN {X 0,Y 558.737,Z 467.282,A -85,B 0,C 180,E1 -2789.278,E2 -2789.278} C_VEL
LIN {X 0,Y 558.738,Z 467.496,A -85,B 0,C 180,E1 -2789.999,E2 -2789.999} C_VEL
LIN {X 0,Y 558.744,Z 466.957,A -85,B 0,C 180,E1 -2791.441,E2 -2791.441} C_VEL
LIN {X 0,Y 558.795,Z 465.245,A -85,B 0,C 180,E1 -2792.883,E2 -2792.883} C_VEL
LIN {X 0,Y 558.819,Z 464.003,A -85,B 0,C 180,E1 -2793.604,E2 -2793.604} C_VEL
LIN {X 0,Y 558.856,Z 459.425,A -85,B 0,C 180,E1 -2795.411,E2 -2795.411} C_VEL
LIN {X 0,Y 558.867,Z 454.479,A -85,B 0,C 180,E1 -2796.824,E2 -2796.824} C_VEL
LIN {X 0,Y 558.969,Z 447.872,A -85,B 0,C 180,E1 -2798.313,E2 -2798.313} C_VEL
LIN {X 0,Y 559.075,Z 439.677,A -85,B 0,C 180,E1 -2799.77,E2 -2799.77} C_VEL
LIN {X 0,Y 559.216,Z 432.304,A -85,B 0,C 180,E1 -2800.865,E2 -2800.865} C_VEL
LIN {X 0,Y 559.312,Z 423.687,A -85,B 0,C 180,E1 -2801.965,E2 -2801.965} C_VEL
LIN {X 0,Y 559.534,Z 415.352,A -85,B 0,C 180,E1 -2802.881,E2 -2802.881} C_VEL
LIN {X 0,Y 559.716,Z 405.737,A -85,B 0,C 180,E1 -2803.801,E2 -2803.801} C_VEL
LIN {X 0,Y 559.973,Z 395.414,A -85,B 0,C 180,E1 -2804.65,E2 -2804.65} C_VEL
LIN {X 0,Y 560.219,Z 382.51,A -85,B 0,C 180,E1 -2805.553,E2 -2805.553} C_VEL
LIN {X 0,Y 560.549,Z 369.431,A -85,B 0,C 180,E1 -2806.291,E2 -2806.291} C_VEL
LIN {X 0,Y 560.702,Z 357.445,A -85,B 0,C 180,E1 -2806.848,E2 -2806.848} C_VEL
LIN {X 0,Y 560.909,Z 344.357,A -85,B 0,C 180,E1 -2807.335,E2 -2807.335} C_VEL
LIN {X 0,Y 561.109,Z 330.942,A -85,B 0,C 180,E1 -2807.713,E2 -2807.713} C_VEL
LIN {X 0,Y 561.264,Z 316.406,A -85,B 0,C 180,E1 -2807.991,E2 -2807.991} C_VEL
LIN {X 0,Y 561.799,Z 165.173,A -85,B 0,C 180,E1 -2809.982,E2 -2809.982} C_VEL
LIN {X 0,Y 560.095,Z 157.609,A -85,B 0,C 180,E1 -2810.149,E2 -2810.149} C_VEL
LIN {X 0,Y 560.376,Z 139.559,A -85,B 0,C 180,E1 -2812.683,E2 -2812.683} C_VEL
LIN {X 0,Y 559.18,Z 132.461,A -85,B 0,C 180,E1 -2813.738,E2 -2813.738} C_VEL
LIN {X 0,Y 559.18,Z 132.456,A -85,B 0,C 180,E1 -2816.096,E2 -2816.096} C_VEL
LIN {X 0,Y 559.16,Z 132.455,A -85,B 0,C 180,E1 -2818.528,E2 -2818.528} C_VEL
LIN {X 0,Y 559.15,Z 132.463,A -85,B 0,C 180,E1 -2821.274,E2 -2821.274} C_VEL
LIN {X 0,Y 559.173,Z 132.455,A -85,B 0,C 180,E1 -2823.95,E2 -2823.95} C_VEL
LIN {X 0,Y 559.164,Z 132.453,A -85,B 0,C 180,E1 -2826.447,E2 -2826.447} C_VEL
LIN {X 0,Y 559.172,Z 132.455,A -85,B 0,C 180,E1 -2828.933,E2 -2828.933} C_VEL
LIN {X 0,Y 559.186,Z 132.454,A -85,B 0,C 180,E1 -2831.766,E2 -2831.766} C_VEL
LIN {X 0,Y 559.133,Z 132.457,A -85,B 0,C 180,E1 -2834.738,E2 -2834.738} C_VEL
LIN {X 0,Y 559.169,Z 132.453,A -85,B 0,C 180,E1 -2837.862,E2 -2837.862} C_VEL
LIN {X 0,Y 559.179,Z 132.451,A -85,B 0,C 180,E1 -2840.134,E2 -2840.134} C_VEL
LIN {X 0,Y 559.139,Z 132.46,A -85,B 0,C 180,E1 -2842.891,E2 -2842.891} C_VEL
LIN {X 0,Y 559.15,Z 132.457,A -85,B 0,C 180,E1 -2845.555,E2 -2845.555} C_VEL
LIN {X 0,Y 559.163,Z 132.453,A -85,B 0,C 180,E1 -2848.137,E2 -2848.137} C_VEL
LIN {X 0,Y 559.149,Z 132.455,A -85,B 0,C 180,E1 -2850.647,E2 -2850.647} C_VEL
LIN {X 0,Y 559.162,Z 132.46,A -85,B 0,C 180,E1 -2853.171,E2 -2853.171} C_VEL
LIN {X 0,Y 559.148,Z 132.456,A -85,B 0,C 180,E1 -2855.494,E2 -2855.494} C_VEL
LIN {X 0,Y 559.167,Z 132.457,A -85,B 0,C 180,E1 -2858.624,E2 -2858.624} C_VEL
LIN {X 0,Y 559.162,Z 132.459,A -85,B 0,C 180,E1 -2860.926,E2 -2860.926} C_VEL
LIN {X 0,Y 559.163,Z 132.453,A -85,B 0,C 180,E1 -2863.948,E2 -2863.948} C_VEL
LIN {X 0,Y 559.165,Z 132.452,A -85,B 0,C 180,E1 -2866.184,E2 -2866.184} C_VEL
LIN {X 0,Y 559.2,Z 132.453,A -85,B 0,C 180,E1 -2869.134,E2 -2869.134} C_VEL
LIN {X 0,Y 559.197,Z 132.448,A -85,B 0,C 180,E1 -2872.053,E2 -2872.053} C_VEL
LIN {X 0,Y 559.25,Z 132.448,A -85,B 0,C 180,E1 -2874.953,E2 -2874.953} C_VEL
LIN {X 0,Y 559.24,Z 132.443,A -85,B 0,C 180,E1 -2877.839,E2 -2877.839} C_VEL
LIN {X 0,Y 559.269,Z 132.445,A -85,B 0,C 180,E1 -2880.72,E2 -2880.72} C_VEL
LIN {X 0,Y 559.235,Z 132.45,A -85,B 0,C 180,E1 -2882.881,E2 -2882.881} C_VEL
LIN {X 0,Y 559.22,Z 132.444,A -85,B 0,C 180,E1 -2885.77,E2 -2885.77} C_VEL
LIN {X 0,Y 559.194,Z 132.457,A -85,B 0,C 180,E1 -2888.674,E2 -2888.674} C_VEL
LIN {X 0,Y 559.198,Z 132.447,A -85,B 0,C 180,E1 -2891.601,E2 -2891.601} C_VEL
LIN {X 0,Y 559.188,Z 132.457,A -85,B 0,C 180,E1 -2894.596,E2 -2894.596} C_VEL
LIN {X 0,Y 559.154,Z 132.453,A -85,B 0,C 180,E1 -2897.557,E2 -2897.557} C_VEL
LIN {X 0,Y 559.165,Z 132.451,A -85,B 0,C 180,E1 -2899.838,E2 -2899.838} C_VEL
LIN {X 0,Y 559.144,Z 132.461,A -85,B 0,C 180,E1 -2902.153,E2 -2902.153} C_VEL
LIN {X 0,Y 559.15,Z 132.46,A -85,B 0,C 180,E1 -2904.505,E2 -2904.505} C_VEL
LIN {X 0,Y 559.162,Z 132.455,A -85,B 0,C 180,E1 -2906.903,E2 -2906.903} C_VEL
LIN {X 0,Y 559.139,Z 132.457,A -85,B 0,C 180,E1 -2909.858,E2 -2909.858} C_VEL
LIN {X 0,Y 559.166,Z 132.455,A -85,B 0,C 180,E1 -2912.715,E2 -2912.715} C_VEL
LIN {X 0,Y 559.149,Z 132.454,A -85,B 0,C 180,E1 -2915.322,E2 -2915.322} C_VEL
LIN {X 0,Y 559.125,Z 132.465,A -85,B 0,C 180,E1 -2918.018,E2 -2918.018} C_VEL
LIN {X 0,Y 559.168,Z 132.448,A -85,B 0,C 180,E1 -2920.811,E2 -2920.811} C_VEL
LIN {X 0,Y 559.133,Z 132.461,A -85,B 0,C 180,E1 -2923.735,E2 -2923.735} C_VEL
LIN {X 0,Y 559.16,Z 132.454,A -85,B 0,C 180,E1 -2926.802,E2 -2926.802} C_VEL
LIN {X 0,Y 559.17,Z 132.453,A -85,B 0,C 180,E1 -2929.19,E2 -2929.19} C_VEL
LIN {X 0,Y 559.128,Z 132.465,A -85,B 0,C 180,E1 -2931.984,E2 -2931.984} C_VEL
LIN {X 0,Y 559.142,Z 132.455,A -85,B 0,C 180,E1 -2934.786,E2 -2934.786} C_VEL
LIN {X 0,Y 559.167,Z 132.455,A -85,B 0,C 180,E1 -2937.363,E2 -2937.363} C_VEL
LIN {X 0,Y 559.181,Z 132.457,A -85,B 0,C 180,E1 -2940.526,E2 -2940.526} C_VEL
LIN {X 0,Y 562.275,Z 143.309,A -85,B 0,C 180,E1 -2941.644,E2 -2941.644} C_VEL
LIN {X 0,Y 561.946,Z 168.047,A -85,B 0,C 180,E1 -2943.743,E2 -2943.743} C_VEL
LIN {X 0,Y 561.376,Z 199.756,A -85,B 0,C 180,E1 -2946.385,E2 -2946.385} C_VEL
LIN {X 0,Y 560.973,Z 233.147,A -85,B 0,C 180,E1 -2949.082,E2 -2949.082} C_VEL
LIN {X 0,Y 560.812,Z 243.144,A -85,B 0,C 180,E1 -2949.881,E2 -2949.881} C_VEL
LIN {X 0,Y 561.812,Z 251.756,A -85,B 0,C 180,E1 -2950.027,E2 -2950.027} C_VEL
LIN {X 0,Y 561.236,Z 412.335,A -85,B 0,C 180,E1 -2952.152,E2 -2952.152} C_VEL
LIN {X 0,Y 561.052,Z 427.74,A -85,B 0,C 180,E1 -2952.505,E2 -2952.505} C_VEL
LIN {X 0,Y 560.842,Z 443.062,A -85,B 0,C 180,E1 -2953.015,E2 -2953.015} C_VEL
LIN {X 0,Y 560.552,Z 456.802,A -85,B 0,C 180,E1 -2953.616,E2 -2953.616} C_VEL
LIN {X 0,Y 560.276,Z 470.269,A -85,B 0,C 180,E1 -2954.355,E2 -2954.355} C_VEL
LIN {X 0,Y 559.995,Z 483.317,A -85,B 0,C 180,E1 -2955.231,E2 -2955.231} C_VEL
LIN {X 0,Y 559.722,Z 495.303,A -85,B 0,C 180,E1 -2956.199,E2 -2956.199} C_VEL
LIN {X 0,Y 559.515,Z 506.758,A -85,B 0,C 180,E1 -2957.303,E2 -2957.303} C_VEL
LIN {X 0,Y 559.302,Z 516.398,A -85,B 0,C 180,E1 -2958.403,E2 -2958.403} C_VEL
LIN {X 0,Y 559.168,Z 525.862,A -85,B 0,C 180,E1 -2959.683,E2 -2959.683} C_VEL
LIN {X 0,Y 559.002,Z 533.742,A -85,B 0,C 180,E1 -2960.959,E2 -2960.959} C_VEL
LIN {X 0,Y 558.919,Z 541.096,A -85,B 0,C 180,E1 -2962.414,E2 -2962.414} C_VEL
LIN {X 0,Y 558.859,Z 546.926,A -85,B 0,C 180,E1 -2963.865,E2 -2963.865} C_VEL
LIN {X 0,Y 558.787,Z 550.388,A -85,B 0,C 180,E1 -2964.95,E2 -2964.95} C_VEL
LIN {X 0,Y 558.818,Z 553.89,A -85,B 0,C 180,E1 -2966.396,E2 -2966.396} C_VEL
LIN {X 0,Y 558.745,Z 556.192,A -85,B 0,C 180,E1 -2967.838,E2 -2967.838} C_VEL
LIN {X 0,Y 558.739,Z 557.349,A -85,B 0,C 180,E1 -2969.28,E2 -2969.28} C_VEL
LIN {X 0,Y 558.739,Z 557.348,A -85,B 0,C 180,E1 -2970.722,E2 -2970.722} C_VEL
LIN {X 0,Y 558.745,Z 556.187,A -85,B 0,C 180,E1 -2972.163,E2 -2972.163} C_VEL
LIN {X 0,Y 558.818,Z 553.883,A -85,B 0,C 180,E1 -2973.606,E2 -2973.606} C_VEL
LIN {X 0,Y 558.787,Z 550.384,A -85,B 0,C 180,E1 -2975.052,E2 -2975.052} C_VEL
LIN {X 0,Y 558.851,Z 545.606,A -85,B 0,C 180,E1 -2976.5,E2 -2976.5} C_VEL
LIN {X 0,Y 558.951,Z 539.417,A -85,B 0,C 180,E1 -2977.951,E2 -2977.951} C_VEL
LIN {X 0,Y 559.005,Z 531.64,A -85,B 0,C 180,E1 -2979.407,E2 -2979.407} C_VEL
LIN {X 0,Y 559.218,Z 523.362,A -85,B 0,C 180,E1 -2980.684,E2 -2980.684} C_VEL
LIN {X 0,Y 559.363,Z 513.385,A -85,B 0,C 180,E1 -2981.966,E2 -2981.966} C_VEL
LIN {X 0,Y 559.597,Z 503.177,A -85,B 0,C 180,E1 -2983.066,E2 -2983.066} C_VEL
LIN {X 0,Y 559.863,Z 491.009,A -85,B 0,C 180,E1 -2984.17,E2 -2984.17} C_VEL
LIN {X 0,Y 560.127,Z 478.673,A -85,B 0,C 180,E1 -2985.101,E2 -2985.101} C_VEL
LIN {X 0,Y 560.39,Z 465.492,A -85,B 0,C 180,E1 -2985.923,E2 -2985.923} C_VEL
LIN {X 0,Y 560.688,Z 450.805,A -85,B 0,C 180,E1 -2986.663,E2 -2986.663} C_VEL
LIN {X 0,Y 560.944,Z 436.591,A -85,B 0,C 180,E1 -2987.218,E2 -2987.218} C_VEL
LIN {X 0,Y 561.121,Z 421.629,A -85,B 0,C 180,E1 -2987.651,E2 -2987.651} C_VEL
LIN {X 0,Y 561.24,Z 406.75,A -85,B 0,C 180,E1 -2987.937,E2 -2987.937} C_VEL
LIN {X 0,Y 561.838,Z 250.469,A -85,B 0,C 180,E1 -2989.989,E2 -2989.989} C_VEL
LIN {X 0,Y 560.792,Z 242.835,A -85,B 0,C 180,E1 -2990.142,E2 -2990.142} C_VEL
LIN {X 0,Y 561.28,Z 205.337,A -85,B 0,C 180,E1 -2993.133,E2 -2993.133} C_VEL
LIN {X 0,Y 561.801,Z 168.481,A -85,B 0,C 180,E1 -2996.166,E2 -2996.166} C_VEL
LIN {X 0,Y 562.18,Z 143.695,A -85,B 0,C 180,E1 -2998.262,E2 -2998.262} C_VEL
LIN {X 0,Y 559.577,Z 134.051,A -85,B 0,C 180,E1 -2999.241,E2 -2999.241} C_VEL
LIN {X 0,Y 559.154,Z 132.462,A -85,B 0,C 180,E1 -2999.436,E2 -2999.436} C_VEL
LIN {X 0,Y 559.164,Z 132.462,A -85,B 0,C 180,E1 -3001.864,E2 -3001.864} C_VEL
LIN {X 0,Y 559.138,Z 132.461,A -85,B 0,C 180,E1 -3004.446,E2 -3004.446} C_VEL
LIN {X 0,Y 559.133,Z 132.466,A -85,B 0,C 180,E1 -3007.639,E2 -3007.639} C_VEL
LIN {X 0,Y 559.152,Z 132.461,A -85,B 0,C 180,E1 -3009.941,E2 -3009.941} C_VEL
LIN {X 0,Y 559.114,Z 132.462,A -85,B 0,C 180,E1 -3012.749,E2 -3012.749} C_VEL
LIN {X 0,Y 559.122,Z 132.463,A -85,B 0,C 180,E1 -3015.765,E2 -3015.765} C_VEL
LIN {X 0,Y 559.091,Z 132.464,A -85,B 0,C 180,E1 -3018.223,E2 -3018.223} C_VEL
LIN {X 0,Y 559.135,Z 132.466,A -85,B 0,C 180,E1 -3021.198,E2 -3021.198} C_VEL
LIN {X 0,Y 559.111,Z 132.462,A -85,B 0,C 180,E1 -3023.787,E2 -3023.787} C_VEL
LIN {X 0,Y 559.139,Z 132.461,A -85,B 0,C 180,E1 -3026.424,E2 -3026.424} C_VEL
LIN {X 0,Y 559.144,Z 132.464,A -85,B 0,C 180,E1 -3028.98,E2 -3028.98} C_VEL
LIN {X 0,Y 559.113,Z 132.463,A -85,B 0,C 180,E1 -3031.63,E2 -3031.63} C_VEL
LIN {X 0,Y 559.161,Z 132.46,A -85,B 0,C 180,E1 -3033.902,E2 -3033.902} C_VEL
LIN {X 0,Y 559.127,Z 132.521,A -85,B 0,C 180,E1 -3036.012,E2 -3036.012} C_VEL
LIN {X 0,Y 560.619,Z 139.146,A -85,B 0,C 180,E1 -3037.131,E2 -3037.131} C_VEL
LIN {X 0,Y 560.428,Z 152.86,A -85,B 0,C 180,E1 -3039.252,E2 -3039.252} C_VEL
LIN {X 0,Y 560.018,Z 171.567,A -85,B 0,C 180,E1 -3042.094,E2 -3042.094} C_VEL
LIN {X 0,Y 559.595,Z 190.01,A -85,B 0,C 180,E1 -3044.913,E2 -3044.913} C_VEL
LIN {X 0,Y 559.522,Z 195.937,A -85,B 0,C 180,E1 -3045.811,E2 -3045.811} C_VEL
LIN {X 0,Y 560.424,Z 201.483,A -85,B 0,C 180,E1 -3045.915,E2 -3045.915} C_VEL
LIN {X 0,Y 560.081,Z 304.066,A -85,B 0,C 180,E1 -3047.292,E2 -3047.292} C_VEL
LIN {X 0,Y 559.986,Z 316.455,A -85,B 0,C 180,E1 -3047.589,E2 -3047.589} C_VEL
LIN {X 0,Y 559.828,Z 329.261,A -85,B 0,C 180,E1 -3048.046,E2 -3048.046} C_VEL
LIN {X 0,Y 559.671,Z 340.839,A -85,B 0,C 180,E1 -3048.607,E2 -3048.607} C_VEL
LIN {X 0,Y 559.456,Z 352.2,A -85,B 0,C 180,E1 -3049.322,E2 -3049.322} C_VEL
LIN {X 0,Y 559.29,Z 362.578,A -85,B 0,C 180,E1 -3050.142,E2 -3050.142} C_VEL
LIN {X 0,Y 559.197,Z 371.175,A -85,B 0,C 180,E1 -3050.961,E2 -3050.961} C_VEL
LIN {X 0,Y 559.051,Z 379.096,A -85,B 0,C 180,E1 -3051.87,E2 -3051.87} C_VEL
LIN {X 0,Y 558.972,Z 386.954,A -85,B 0,C 180,E1 -3052.977,E2 -3052.977} C_VEL
LIN {X 0,Y 558.936,Z 393.953,A -85,B 0,C 180,E1 -3054.227,E2 -3054.227} C_VEL
LIN {X 0,Y 558.827,Z 398.696,A -85,B 0,C 180,E1 -3055.311,E2 -3055.311} C_VEL
LIN {X 0,Y 558.837,Z 402.327,A -85,B 0,C 180,E1 -3056.395,E2 -3056.395} C_VEL
LIN {X 0,Y 558.799,Z 404.204,A -85,B 0,C 180,E1 -3057.116,E2 -3057.116} C_VEL
LIN {X 0,Y 558.745,Z 405.625,A -85,B 0,C 180,E1 -3057.838,E2 -3057.838} C_VEL
LIN {X 0,Y 558.742,Z 407.256,A -85,B 0,C 180,E1 -3059.279,E2 -3059.279} C_VEL
LIN {X 0,Y 558.74,Z 407.496,A -85,B 0,C 180,E1 -3060,E2 -3060} C_VEL
LIN {X 0,Y 558.741,Z 407.316,A -85,B 0,C 180,E1 -3060.721,E2 -3060.721} C_VEL
LIN {X 0,Y 558.745,Z 405.768,A -85,B 0,C 180,E1 -3062.163,E2 -3062.163} C_VEL
LIN {X 0,Y 558.8,Z 404.407,A -85,B 0,C 180,E1 -3062.884,E2 -3062.884} C_VEL
LIN {X 0,Y 558.844,Z 401.526,A -85,B 0,C 180,E1 -3063.966,E2 -3063.966} C_VEL
LIN {X 0,Y 558.798,Z 397.625,A -85,B 0,C 180,E1 -3065.051,E2 -3065.051} C_VEL
LIN {X 0,Y 558.91,Z 392.597,A -85,B 0,C 180,E1 -3066.136,E2 -3066.136} C_VEL
LIN {X 0,Y 558.973,Z 386.266,A -85,B 0,C 180,E1 -3067.223,E2 -3067.223} C_VEL
LIN {X 0,Y 559.091,Z 378.343,A -85,B 0,C 180,E1 -3068.312,E2 -3068.312} C_VEL
LIN {X 0,Y 559.223,Z 368.489,A -85,B 0,C 180,E1 -3069.403,E2 -3069.403} C_VEL
LIN {X 0,Y 559.41,Z 358.171,A -85,B 0,C 180,E1 -3070.313,E2 -3070.313} C_VEL
LIN {X 0,Y 559.582,Z 347.172,A -85,B 0,C 180,E1 -3071.099,E2 -3071.099} C_VEL
LIN {X 0,Y 559.737,Z 335.141,A -85,B 0,C 180,E1 -3071.773,E2 -3071.773} C_VEL
LIN {X 0,Y 559.809,Z 323.16,A -85,B 0,C 180,E1 -3072.277,E2 -3072.277} C_VEL
LIN {X 0,Y 559.97,Z 310.123,A -85,B 0,C 180,E1 -3072.665,E2 -3072.665} C_VEL
LIN {X 0,Y 560.089,Z 297.728,A -85,B 0,C 180,E1 -3072.892,E2 -3072.892} C_VEL
LIN {X 0,Y 560.195,Z 200.671,A -85,B 0,C 180,E1 -3074.153,E2 -3074.153} C_VEL
LIN {X 0,Y 559.431,Z 195.602,A -85,B 0,C 180,E1 -3074.25,E2 -3074.25} C_VEL
LIN {X 0,Y 559.557,Z 182.779,A -85,B 0,C 180,E1 -3076.144,E2 -3076.144} C_VEL
LIN {X 0,Y 558.953,Z 179.568,A -85,B 0,C 180,E1 -3076.647,E2 -3076.647} C_VEL
LIN {X 0,Y 553.553,Z 169.718,A -85,B 0,C 180,E1 -3078.336,E2 -3078.336} C_VEL
LIN {X 0,Y 552.939,Z 166.484,A -85,B 0,C 180,E1 -3078.847,E2 -3078.847} C_VEL
LIN {X 0,Y 553.236,Z 149.428,A -85,B 0,C 180,E1 -3081.421,E2 -3081.421} C_VEL
LIN {X 0,Y 553.449,Z 140.433,A -85,B 0,C 180,E1 -3082.787,E2 -3082.787} C_VEL
LIN {X 0,Y 552.14,Z 133.336,A -85,B 0,C 180,E1 -3083.975,E2 -3083.975} C_VEL
LIN {X 0,Y 552.092,Z 133.336,A -85,B 0,C 180,E1 -3086.458,E2 -3086.458} C_VEL
LIN {X 0,Y 552.097,Z 133.337,A -85,B 0,C 180,E1 -3088.929,E2 -3088.929} C_VEL
LIN {X 0,Y 552.116,Z 133.34,A -85,B 0,C 180,E1 -3091.475,E2 -3091.475} C_VEL
LIN {X 0,Y 552.135,Z 133.329,A -85,B 0,C 180,E1 -3094.17,E2 -3094.17} C_VEL
LIN {X 0,Y 552.103,Z 133.335,A -85,B 0,C 180,E1 -3096.747,E2 -3096.747} C_VEL
LIN {X 0,Y 552.133,Z 133.331,A -85,B 0,C 180,E1 -3099.527,E2 -3099.527} C_VEL
LIN {X 0,Y 552.112,Z 133.333,A -85,B 0,C 180,E1 -3102.427,E2 -3102.427} C_VEL
LIN {X 0,Y 552.099,Z 133.336,A -85,B 0,C 180,E1 -3105.562,E2 -3105.562} C_VEL
LIN {X 0,Y 552.125,Z 133.334,A -85,B 0,C 180,E1 -3108.554,E2 -3108.554} C_VEL
LIN {X 0,Y 552.12,Z 133.334,A -85,B 0,C 180,E1 -3111.41,E2 -3111.41} C_VEL
LIN {X 0,Y 552.089,Z 133.337,A -85,B 0,C 180,E1 -3114.156,E2 -3114.156} C_VEL
LIN {X 0,Y 552.111,Z 133.34,A -85,B 0,C 180,E1 -3116.813,E2 -3116.813} C_VEL
LIN {X 0,Y 552.103,Z 133.335,A -85,B 0,C 180,E1 -3119.39,E2 -3119.39} C_VEL
LIN {X 0,Y 552.097,Z 133.336,A -85,B 0,C 180,E1 -3121.9,E2 -3121.9} C_VEL
LIN {X 0,Y 552.16,Z 133.335,A -85,B 0,C 180,E1 -3124.649,E2 -3124.649} C_VEL
LIN {X 0,Y 552.139,Z 133.447,A -85,B 0,C 180,E1 -3126.156,E2 -3126.156} C_VEL
LIN {X 0,Y 553.493,Z 140.435,A -85,B 0,C 180,E1 -3127.214,E2 -3127.214} C_VEL
LIN {X 0,Y 553.265,Z 157.926,A -85,B 0,C 180,E1 -3129.67,E2 -3129.67} C_VEL
LIN {X 0,Y 555.186,Z 167.265,A -85,B 0,C 180,E1 -3129.883,E2 -3129.883} C_VEL
LIN {X 0,Y 554.487,Z 322.626,A -85,B 0,C 180,E1 -3131.97,E2 -3131.97} C_VEL
LIN {X 0,Y 554.326,Z 337.382,A -85,B 0,C 180,E1 -3132.308,E2 -3132.308} C_VEL
LIN {X 0,Y 554.053,Z 352.295,A -85,B 0,C 180,E1 -3132.799,E2 -3132.799} C_VEL
LIN {X 0,Y 553.817,Z 366.212,A -85,B 0,C 180,E1 -3133.409,E2 -3133.409} C_VEL
LIN {X 0,Y 553.463,Z 379.774,A -85,B 0,C 180,E1 -3134.156,E2 -3134.156} C_VEL
LIN {X 0,Y 553.086,Z 393.752,A -85,B 0,C 180,E1 -3135.109,E2 -3135.109} C_VEL
LIN {X 0,Y 552.793,Z 404.738,A -85,B 0,C 180,E1 -3136.021,E2 -3136.021} C_VEL
LIN {X 0,Y 552.563,Z 414.459,A -85,B 0,C 180,E1 -3136.952,E2 -3136.952} C_VEL
LIN {X 0,Y 552.354,Z 422.903,A -85,B 0,C 180,E1 -3137.88,E2 -3137.88} C_VEL
LIN {X 0,Y 552.174,Z 430.47,A -85,B 0,C 180,E1 -3138.834,E2 -3138.834} C_VEL
LIN {X 0,Y 552.066,Z 437.916,A -85,B 0,C 180,E1 -3139.918,E2 -3139.918} C_VEL
LIN {X 0,Y 551.922,Z 444.443,A -85,B 0,C 180,E1 -3141.025,E2 -3141.025} C_VEL
LIN {X 0,Y 551.876,Z 449.157,A -85,B 0,C 180,E1 -3141.947,E2 -3141.947} C_VEL
LIN {X 0,Y 551.814,Z 453.98,A -85,B 0,C 180,E1 -3143.05,E2 -3143.05} C_VEL
LIN {X 0,Y 551.786,Z 459.132,A -85,B 0,C 180,E1 -3144.518,E2 -3144.518} C_VEL
LIN {X 0,Y 551.73,Z 463.825,A -85,B 0,C 180,E1 -3146.347,E2 -3146.347} C_VEL
LIN {X 0,Y 551.655,Z 466.128,A -85,B 0,C 180,E1 -3147.809,E2 -3147.809} C_VEL
LIN {X 0,Y 551.637,Z 467.275,A -85,B 0,C 180,E1 -3149.269,E2 -3149.269} C_VEL
LIN {X 0,Y 551.638,Z 467.496,A -85,B 0,C 180,E1 -3149.999,E2 -3149.999} C_VEL
LIN {X 0,Y 551.644,Z 466.95,A -85,B 0,C 180,E1 -3151.459,E2 -3151.459} C_VEL
LIN {X 0,Y 551.719,Z 465.236,A -85,B 0,C 180,E1 -3152.92,E2 -3152.92} C_VEL
LIN {X 0,Y 551.731,Z 464.005,A -85,B 0,C 180,E1 -3153.651,E2 -3153.651} C_VEL
LIN {X 0,Y 551.785,Z 459.415,A -85,B 0,C 180,E1 -3155.481,E2 -3155.481} C_VEL
LIN {X 0,Y 551.78,Z 455.732,A -85,B 0,C 180,E1 -3156.581,E2 -3156.581} C_VEL
LIN {X 0,Y 551.83,Z 451.27,A -85,B 0,C 180,E1 -3157.684,E2 -3157.684} C_VEL
LIN {X 0,Y 551.917,Z 445.941,A -85,B 0,C 180,E1 -3158.789,E2 -3158.789} C_VEL
LIN {X 0,Y 552.014,Z 439.663,A -85,B 0,C 180,E1 -3159.896,E2 -3159.896} C_VEL
LIN {X 0,Y 552.171,Z 432.292,A -85,B 0,C 180,E1 -3161.005,E2 -3161.005} C_VEL
LIN {X 0,Y 552.288,Z 425.225,A -85,B 0,C 180,E1 -3161.933,E2 -3161.933} C_VEL
LIN {X 0,Y 552.51,Z 417.122,A -85,B 0,C 180,E1 -3162.861,E2 -3162.861} C_VEL
LIN {X 0,Y 552.702,Z 407.768,A -85,B 0,C 180,E1 -3163.792,E2 -3163.792} C_VEL
LIN {X 0,Y 553.059,Z 395.972,A -85,B 0,C 180,E1 -3164.808,E2 -3164.808} C_VEL
LIN {X 0,Y 553.368,Z 382.759,A -85,B 0,C 180,E1 -3165.751,E2 -3165.751} C_VEL
LIN {X 0,Y 553.764,Z 369.916,A -85,B 0,C 180,E1 -3166.496,E2 -3166.496} C_VEL
LIN {X 0,Y 553.988,Z 355.874,A -85,B 0,C 180,E1 -3167.154,E2 -3167.154} C_VEL
LIN {X 0,Y 554.275,Z 340.66,A -85,B 0,C 180,E1 -3167.692,E2 -3167.692} C_VEL
LIN {X 0,Y 554.465,Z 325.12,A -85,B 0,C 180,E1 -3168.076,E2 -3168.076} C_VEL
LIN {X 0,Y 554.601,Z 299.539,A -85,B 0,C 180,E1 -3168.448,E2 -3168.448} C_VEL
LIN {X 0,Y 555.193,Z 166.618,A -85,B 0,C 180,E1 -3170.216,E2 -3170.216} C_VEL
LIN {X 0,Y 553.248,Z 157.87,A -85,B 0,C 180,E1 -3170.431,E2 -3170.431} C_VEL
LIN {X 0,Y 553.53,Z 141.118,A -85,B 0,C 180,E1 -3172.782,E2 -3172.782} C_VEL
LIN {X 0,Y 552.518,Z 135.159,A -85,B 0,C 180,E1 -3173.675,E2 -3173.675} C_VEL
LIN {X 0,Y 552.137,Z 133.337,A -85,B 0,C 180,E1 -3173.974,E2 -3173.974} C_VEL
LIN {X 0,Y 552.118,Z 133.334,A -85,B 0,C 180,E1 -3176.455,E2 -3176.455} C_VEL
LIN {X 0,Y 552.107,Z 133.335,A -85,B 0,C 180,E1 -3178.927,E2 -3178.927} C_VEL
LIN {X 0,Y 552.132,Z 133.336,A -85,B 0,C 180,E1 -3181.479,E2 -3181.479} C_VEL
LIN {X 0,Y 552.141,Z 133.329,A -85,B 0,C 180,E1 -3184.171,E2 -3184.171} C_VEL
LIN {X 0,Y 552.107,Z 133.333,A -85,B 0,C 180,E1 -3186.745,E2 -3186.745} C_VEL
LIN {X 0,Y 552.128,Z 133.331,A -85,B 0,C 180,E1 -3189.526,E2 -3189.526} C_VEL
LIN {X 0,Y 552.125,Z 133.33,A -85,B 0,C 180,E1 -3192.424,E2 -3192.424} C_VEL
LIN {X 0,Y 552.091,Z 133.34,A -85,B 0,C 180,E1 -3195.562,E2 -3195.562} C_VEL
LIN {X 0,Y 552.133,Z 133.33,A -85,B 0,C 180,E1 -3198.675,E2 -3198.675} C_VEL
LIN {X 0,Y 552.113,Z 133.337,A -85,B 0,C 180,E1 -3201.41,E2 -3201.41} C_VEL
LIN {X 0,Y 552.106,Z 133.332,A -85,B 0,C 180,E1 -3204.158,E2 -3204.158} C_VEL
LIN {X 0,Y 552.114,Z 133.334,A -85,B 0,C 180,E1 -3206.814,E2 -3206.814} C_VEL
LIN {X 0,Y 552.106,Z 133.334,A -85,B 0,C 180,E1 -3209.391,E2 -3209.391} C_VEL
LIN {X 0,Y 552.117,Z 133.331,A -85,B 0,C 180,E1 -3211.902,E2 -3211.902} C_VEL
LIN {X 0,Y 552.145,Z 133.33,A -85,B 0,C 180,E1 -3214.649,E2 -3214.649} C_VEL
LIN {X 0,Y 552.087,Z 133.337,A -85,B 0,C 180,E1 -3217.549,E2 -3217.549} C_VEL
LIN {X 0,Y 552.139,Z 133.328,A -85,B 0,C 180,E1 -3220.373,E2 -3220.373} C_VEL
LIN {X 0,Y 552.148,Z 133.336,A -85,B 0,C 180,E1 -3222.977,E2 -3222.977} C_VEL
LIN {X 0,Y 552.127,Z 133.328,A -85,B 0,C 180,E1 -3226.004,E2 -3226.004} C_VEL
LIN {X 0,Y 552.168,Z 133.332,A -85,B 0,C 180,E1 -3228.993,E2 -3228.993} C_VEL
LIN {X 0,Y 552.151,Z 133.326,A -85,B 0,C 180,E1 -3231.951,E2 -3231.951} C_VEL
LIN {X 0,Y 552.224,Z 133.325,A -85,B 0,C 180,E1 -3234.889,E2 -3234.889} C_VEL
LIN {X 0,Y 552.212,Z 133.319,A -85,B 0,C 180,E1 -3237.812,E2 -3237.812} C_VEL
LIN {X 0,Y 552.238,Z 133.32,A -85,B 0,C 180,E1 -3240.729,E2 -3240.729} C_VEL
LIN {X 0,Y 552.201,Z 133.325,A -85,B 0,C 180,E1 -3242.918,E2 -3242.918} C_VEL
LIN {X 0,Y 552.19,Z 133.32,A -85,B 0,C 180,E1 -3245.844,E2 -3245.844} C_VEL
LIN {X 0,Y 552.161,Z 133.331,A -85,B 0,C 180,E1 -3248.786,E2 -3248.786} C_VEL
LIN {X 0,Y 552.154,Z 133.324,A -85,B 0,C 180,E1 -3251.751,E2 -3251.751} C_VEL
LIN {X 0,Y 552.125,Z 133.334,A -85,B 0,C 180,E1 -3254.749,E2 -3254.749} C_VEL
LIN {X 0,Y 552.105,Z 133.331,A -85,B 0,C 180,E1 -3257.789,E2 -3257.789} C_VEL
LIN {X 0,Y 552.124,Z 133.331,A -85,B 0,C 180,E1 -3260.101,E2 -3260.101} C_VEL
LIN {X 0,Y 552.103,Z 133.34,A -85,B 0,C 180,E1 -3262.45,E2 -3262.45} C_VEL
LIN {X 0,Y 552.144,Z 133.325,A -85,B 0,C 180,E1 -3265.351,E2 -3265.351} C_VEL
LIN {X 0,Y 552.117,Z 133.337,A -85,B 0,C 180,E1 -3268.098,E2 -3268.098} C_VEL
LIN {X 0,Y 552.098,Z 133.337,A -85,B 0,C 180,E1 -3270.609,E2 -3270.609} C_VEL
LIN {X 0,Y 552.114,Z 133.33,A -85,B 0,C 180,E1 -3273.186,E2 -3273.186} C_VEL
LIN {X 0,Y 552.104,Z 133.336,A -85,B 0,C 180,E1 -3275.842,E2 -3275.842} C_VEL
LIN {X 0,Y 552.114,Z 133.326,A -85,B 0,C 180,E1 -3279.062,E2 -3279.062} C_VEL
LIN {X 0,Y 552.131,Z 133.324,A -85,B 0,C 180,E1 -3281.445,E2 -3281.445} C_VEL
LIN {X 0,Y 552.087,Z 133.338,A -85,B 0,C 180,E1 -3284.533,E2 -3284.533} C_VEL
LIN {X 0,Y 552.123,Z 133.333,A -85,B 0,C 180,E1 -3287.585,E2 -3287.585} C_VEL
LIN {X 0,Y 552.127,Z 133.332,A -85,B 0,C 180,E1 -3290.474,E2 -3290.474} C_VEL
LIN {X 0,Y 552.108,Z 133.332,A -85,B 0,C 180,E1 -3293.317,E2 -3293.317} C_VEL
LIN {X 0,Y 552.122,Z 133.336,A -85,B 0,C 180,E1 -3295.94,E2 -3295.94} C_VEL
LIN {X 0,Y 552.114,Z 133.336,A -85,B 0,C 180,E1 -3298.542,E2 -3298.542} C_VEL
LIN {X 0,Y 552.127,Z 133.4,A -85,B 0,C 180,E1 -3300.237,E2 -3300.237} C_VEL
LIN {X 0,Y 555.61,Z 145.257,A -85,B 0,C 180,E1 -3301.479,E2 -3301.479} C_VEL
LIN {X 0,Y 555.249,Z 167.529,A -85,B 0,C 180,E1 -3303.402,E2 -3303.402} C_VEL
LIN {X 0,Y 554.584,Z 200.366,A -85,B 0,C 180,E1 -3306.177,E2 -3306.177} C_VEL
LIN {X 0,Y 554.057,Z 234.902,A -85,B 0,C 180,E1 -3309.003,E2 -3309.003} C_VEL
LIN {X 0,Y 553.917,Z 243.001,A -85,B 0,C 180,E1 -3309.663,E2 -3309.663} C_VEL
LIN {X 0,Y 555.023,Z 251.93,A -85,B 0,C 180,E1 -3309.819,E2 -3309.819} C_VEL
LIN {X 0,Y 554.463,Z 412.546,A -85,B 0,C 180,E1 -3311.939,E2 -3311.939} C_VEL
LIN {X 0,Y 554.282,Z 427.645,A -85,B 0,C 180,E1 -3312.285,E2 -3312.285} C_VEL
LIN {X 0,Y 554.041,Z 443.059,A -85,B 0,C 180,E1 -3312.801,E2 -3312.801} C_VEL
LIN {X 0,Y 553.717,Z 456.805,A -85,B 0,C 180,E1 -3313.408,E2 -3313.408} C_VEL
LIN {X 0,Y 553.414,Z 470.271,A -85,B 0,C 180,E1 -3314.156,E2 -3314.156} C_VEL
LIN {X 0,Y 553.075,Z 484.16,A -85,B 0,C 180,E1 -3315.104,E2 -3315.104} C_VEL
LIN {X 0,Y 552.759,Z 496.366,A -85,B 0,C 180,E1 -3316.115,E2 -3316.115} C_VEL
LIN {X 0,Y 552.48,Z 508.519,A -85,B 0,C 180,E1 -3317.325,E2 -3317.325} C_VEL
LIN {X 0,Y 552.214,Z 518.49,A -85,B 0,C 180,E1 -3318.514,E2 -3318.514} C_VEL
LIN {X 0,Y 552.124,Z 527.091,A -85,B 0,C 180,E1 -3319.736,E2 -3319.736} C_VEL
LIN {X 0,Y 551.92,Z 534.748,A -85,B 0,C 180,E1 -3321.027,E2 -3321.027} C_VEL
LIN {X 0,Y 551.836,Z 541.095,A -85,B 0,C 180,E1 -3322.316,E2 -3322.316} C_VEL
LIN {X 0,Y 551.768,Z 546.573,A -85,B 0,C 180,E1 -3323.681,E2 -3323.681} C_VEL
LIN {X 0,Y 551.713,Z 550.388,A -85,B 0,C 180,E1 -3324.885,E2 -3324.885} C_VEL
LIN {X 0,Y 551.73,Z 553.89,A -85,B 0,C 180,E1 -3326.349,E2 -3326.349} C_VEL
LIN {X 0,Y 551.655,Z 556.191,A -85,B 0,C 180,E1 -3327.811,E2 -3327.811} C_VEL
LIN {X 0,Y 551.639,Z 557.348,A -85,B 0,C 180,E1 -3329.271,E2 -3329.271} C_VEL
LIN {X 0,Y 551.639,Z 557.347,A -85,B 0,C 180,E1 -3330.731,E2 -3330.731} C_VEL
LIN {X 0,Y 551.655,Z 556.186,A -85,B 0,C 180,E1 -3332.191,E2 -3332.191} C_VEL
LIN {X 0,Y 551.73,Z 553.882,A -85,B 0,C 180,E1 -3333.653,E2 -3333.653} C_VEL
LIN {X 0,Y 551.713,Z 550.384,A -85,B 0,C 180,E1 -3335.117,E2 -3335.117} C_VEL
LIN {X 0,Y 551.781,Z 545.606,A -85,B 0,C 180,E1 -3336.583,E2 -3336.583} C_VEL
LIN {X 0,Y 551.877,Z 539.417,A -85,B 0,C 180,E1 -3338.053,E2 -3338.053} C_VEL
LIN {X 0,Y 551.951,Z 531.639,A -85,B 0,C 180,E1 -3339.529,E2 -3339.529} C_VEL
LIN {X 0,Y 552.185,Z 523.361,A -85,B 0,C 180,E1 -3340.821,E2 -3340.821} C_VEL
LIN {X 0,Y 552.354,Z 513.385,A -85,B 0,C 180,E1 -3342.12,E2 -3342.12} C_VEL
LIN {X 0,Y 552.609,Z 503.176,A -85,B 0,C 180,E1 -3343.234,E2 -3343.234} C_VEL
LIN {X 0,Y 552.909,Z 491.008,A -85,B 0,C 180,E1 -3344.352,E2 -3344.352} C_VEL
LIN {X 0,Y 553.251,Z 478.426,A -85,B 0,C 180,E1 -3345.311,E2 -3345.311} C_VEL
LIN {X 0,Y 553.54,Z 465.489,A -85,B 0,C 180,E1 -3346.126,E2 -3346.126} C_VEL
LIN {X 0,Y 553.833,Z 450.802,A -85,B 0,C 180,E1 -3346.875,E2 -3346.875} C_VEL
LIN {X 0,Y 554.173,Z 436.58,A -85,B 0,C 180,E1 -3347.435,E2 -3347.435} C_VEL
LIN {X 0,Y 554.34,Z 421.601,A -85,B 0,C 180,E1 -3347.87,E2 -3347.87} C_VEL
LIN {X 0,Y 554.467,Z 406.844,A -85,B 0,C 180,E1 -3348.151,E2 -3348.151} C_VEL
LIN {X 0,Y 554.953,Z 250.344,A -85,B 0,C 180,E1 -3350.194,E2 -3350.194} C_VEL
LIN {X 0,Y 553.887,Z 242.59,A -85,B 0,C 180,E1 -3350.351,E2 -3350.351} C_VEL
LIN {X 0,Y 554.413,Z 205.673,A -85,B 0,C 180,E1 -3353.338,E2 -3353.338} C_VEL
LIN {X 0,Y 555.059,Z 168.914,A -85,B 0,C 180,E1 -3356.408,E2 -3356.408} C_VEL
LIN {X 0,Y 555.51,Z 145.545,A -85,B 0,C 180,E1 -3358.426,E2 -3358.426} C_VEL
LIN {X 0,Y 552.101,Z 133.341,A -85,B 0,C 180,E1 -3359.74,E2 -3359.74} C_VEL
LIN {X 0,Y 552.115,Z 133.339,A -85,B 0,C 180,E1 -3362.319,E2 -3362.319} C_VEL
LIN {X 0,Y 552.079,Z 133.339,A -85,B 0,C 180,E1 -3364.95,E2 -3364.95} C_VEL
LIN {X 0,Y 552.091,Z 133.342,A -85,B 0,C 180,E1 -3367.885,E2 -3367.885} C_VEL
LIN {X 0,Y 552.086,Z 133.337,A -85,B 0,C 180,E1 -3370.484,E2 -3370.484} C_VEL
LIN {X 0,Y 552.062,Z 133.347,A -85,B 0,C 180,E1 -3373.478,E2 -3373.478} C_VEL
LIN {X 0,Y 552.075,Z 133.339,A -85,B 0,C 180,E1 -3376.573,E2 -3376.573} C_VEL
LIN {X 0,Y 552.041,Z 133.347,A -85,B 0,C 180,E1 -3379.513,E2 -3379.513} C_VEL
LIN {X 0,Y 552.07,Z 133.339,A -85,B 0,C 180,E1 -3382.334,E2 -3382.334} C_VEL
LIN {X 0,Y 552.073,Z 133.345,A -85,B 0,C 180,E1 -3385.05,E2 -3385.05} C_VEL
LIN {X 0,Y 552.099,Z 133.337,A -85,B 0,C 180,E1 -3387.68,E2 -3387.68} C_VEL
LIN {X 0,Y 552.078,Z 133.341,A -85,B 0,C 180,E1 -3390.233,E2 -3390.233} C_VEL
LIN {X 0,Y 552.097,Z 133.342,A -85,B 0,C 180,E1 -3393.01,E2 -3393.01} C_VEL
LIN {X 0,Y 552.094,Z 133.375,A -85,B 0,C 180,E1 -3395.712,E2 -3395.712} C_VEL
LIN {X 0,Y 553.843,Z 141.032,A -85,B 0,C 180,E1 -3397.033,E2 -3397.033} C_VEL
LIN {X 0,Y 553.605,Z 154.79,A -85,B 0,C 180,E1 -3399.178,E2 -3399.178} C_VEL
LIN {X 0,Y 553.158,Z 173.52,A -85,B 0,C 180,E1 -3402.055,E2 -3402.055} C_VEL
LIN {X 0,Y 552.698,Z 192.172,A -85,B 0,C 180,E1 -3404.928,E2 -3404.928} C_VEL
LIN {X 0,Y 552.682,Z 196.645,A -85,B 0,C 180,E1 -3405.586,E2 -3405.586} C_VEL
LIN {X 0,Y 553.641,Z 202.015,A -85,B 0,C 180,E1 -3405.694,E2 -3405.694} C_VEL
LIN {X 0,Y 553.178,Z 305.109,A -85,B 0,C 180,E1 -3407.131,E2 -3407.131} C_VEL
LIN {X 0,Y 553.087,Z 318.157,A -85,B 0,C 180,E1 -3407.455,E2 -3407.455} C_VEL
LIN {X 0,Y 552.958,Z 330.162,A -85,B 0,C 180,E1 -3407.895,E2 -3407.895} C_VEL
LIN {X 0,Y 552.736,Z 342.409,A -85,B 0,C 180,E1 -3408.501,E2 -3408.501} C_VEL
LIN {X 0,Y 552.562,Z 353.12,A -85,B 0,C 180,E1 -3409.187,E2 -3409.187} C_VEL
LIN {X 0,Y 552.357,Z 363.509,A -85,B 0,C 180,E1 -3410.017,E2 -3410.017} C_VEL
LIN {X 0,Y 552.244,Z 371.975,A -85,B 0,C 180,E1 -3410.847,E2 -3410.847} C_VEL
LIN {X 0,Y 552.067,Z 379.769,A -85,B 0,C 180,E1 -3411.766,E2 -3411.766} C_VEL
LIN {X 0,Y 551.944,Z 387.477,A -85,B 0,C 180,E1 -3412.887,E2 -3412.887} C_VEL
LIN {X 0,Y 551.868,Z 394.309,A -85,B 0,C 180,E1 -3414.153,E2 -3414.153} C_VEL
LIN {X 0,Y 551.764,Z 398.94,A -85,B 0,C 180,E1 -3415.251,E2 -3415.251} C_VEL
LIN {X 0,Y 551.751,Z 402.469,A -85,B 0,C 180,E1 -3416.349,E2 -3416.349} C_VEL
LIN {X 0,Y 551.724,Z 404.294,A -85,B 0,C 180,E1 -3417.079,E2 -3417.079} C_VEL
LIN {X 0,Y 551.656,Z 405.681,A -85,B 0,C 180,E1 -3417.81,E2 -3417.81} C_VEL
LIN {X 0,Y 551.643,Z 407.261,A -85,B 0,C 180,E1 -3419.27,E2 -3419.27} C_VEL
LIN {X 0,Y 551.641,Z 407.496,A -85,B 0,C 180,E1 -3420,E2 -3420} C_VEL
LIN {X 0,Y 551.646,Z 406.746,A -85,B 0,C 180,E1 -3421.46,E2 -3421.46} C_VEL
LIN {X 0,Y 551.725,Z 404.466,A -85,B 0,C 180,E1 -3422.921,E2 -3422.921} C_VEL
LIN {X 0,Y 551.764,Z 401.652,A -85,B 0,C 180,E1 -3424.017,E2 -3424.017} C_VEL
LIN {X 0,Y 551.724,Z 397.845,A -85,B 0,C 180,E1 -3425.116,E2 -3425.116} C_VEL
LIN {X 0,Y 551.856,Z 392.209,A -85,B 0,C 180,E1 -3426.348,E2 -3426.348} C_VEL
LIN {X 0,Y 551.932,Z 385.463,A -85,B 0,C 180,E1 -3427.5,E2 -3427.5} C_VEL
LIN {X 0,Y 552.1,Z 377.391,A -85,B 0,C 180,E1 -3428.602,E2 -3428.602} C_VEL
LIN {X 0,Y 552.255,Z 369.093,A -85,B 0,C 180,E1 -3429.523,E2 -3429.523} C_VEL
LIN {X 0,Y 552.474,Z 358.831,A -85,B 0,C 180,E1 -3430.444,E2 -3430.444} C_VEL
LIN {X 0,Y 552.657,Z 348.044,A -85,B 0,C 180,E1 -3431.223,E2 -3431.223} C_VEL
LIN {X 0,Y 552.803,Z 336.722,A -85,B 0,C 180,E1 -3431.871,E2 -3431.871} C_VEL
LIN {X 0,Y 552.875,Z 324.956,A -85,B 0,C 180,E1 -3432.387,E2 -3432.387} C_VEL
LIN {X 0,Y 553.087,Z 311.479,A -85,B 0,C 180,E1 -3432.802,E2 -3432.802} C_VEL
LIN {X 0,Y 553.189,Z 298.103,A -85,B 0,C 180,E1 -3433.056,E2 -3433.056} C_VEL
LIN {X 0,Y 553.43,Z 202.037,A -85,B 0,C 180,E1 -3434.328,E2 -3434.328} C_VEL
LIN {X 0,Y 552.469,Z 195.878,A -85,B 0,C 180,E1 -3434.446,E2 -3434.446} C_VEL
LIN {X 0,Y 552.755,Z 175.316,A -85,B 0,C 180,E1 -3437.523,E2 -3437.523} C_VEL
LIN {X 0,Y 552.939,Z 166.484,A -85,B 0,C 180,E1 -3438.847,E2 -3438.847} C_VEL
LIN {X 0,Y 552.323,Z 163.271,A -85,B 0,C 180,E1 -3439.357,E2 -3439.357} C_VEL
LIN {X 0,Y 546.953,Z 153.556,A -85,B 0,C 180,E1 -3441.076,E2 -3441.076} C_VEL
LIN {X 0,Y 546.372,Z 150.344,A -85,B 0,C 180,E1 -3441.595,E2 -3441.595} C_VEL
LIN {X 0,Y 546.573,Z 141.861,A -85,B 0,C 180,E1 -3442.89,E2 -3442.89} C_VEL
LIN {X 0,Y 545.083,Z 134.214,A -85,B 0,C 180,E1 -3444.163,E2 -3444.163} C_VEL
LIN {X 0,Y 545.061,Z 134.213,A -85,B 0,C 180,E1 -3446.826,E2 -3446.826} C_VEL
LIN {X 0,Y 545.059,Z 134.218,A -85,B 0,C 180,E1 -3449.339,E2 -3449.339} C_VEL
LIN {X 0,Y 545.059,Z 134.213,A -85,B 0,C 180,E1 -3451.915,E2 -3451.915} C_VEL
LIN {X 0,Y 545.065,Z 134.21,A -85,B 0,C 180,E1 -3454.564,E2 -3454.564} C_VEL
LIN {X 0,Y 545.036,Z 134.222,A -85,B 0,C 180,E1 -3457.304,E2 -3457.304} C_VEL
LIN {X 0,Y 545.069,Z 134.207,A -85,B 0,C 180,E1 -3460.142,E2 -3460.142} C_VEL
LIN {X 0,Y 545.05,Z 134.218,A -85,B 0,C 180,E1 -3463.11,E2 -3463.11} C_VEL
LIN {X 0,Y 545.054,Z 134.211,A -85,B 0,C 180,E1 -3466.226,E2 -3466.226} C_VEL
LIN {X 0,Y 545.086,Z 134.216,A -85,B 0,C 180,E1 -3468.885,E2 -3468.885} C_VEL
LIN {X 0,Y 545.052,Z 134.212,A -85,B 0,C 180,E1 -3471.864,E2 -3471.864} C_VEL
LIN {X 0,Y 545.04,Z 134.219,A -85,B 0,C 180,E1 -3474.531,E2 -3474.531} C_VEL
LIN {X 0,Y 545.069,Z 134.213,A -85,B 0,C 180,E1 -3477.211,E2 -3477.211} C_VEL
LIN {X 0,Y 545.066,Z 134.211,A -85,B 0,C 180,E1 -3479.81,E2 -3479.81} C_VEL
LIN {X 0,Y 545.089,Z 134.215,A -85,B 0,C 180,E1 -3482.828,E2 -3482.828} C_VEL
LIN {X 0,Y 545.061,Z 134.216,A -85,B 0,C 180,E1 -3485.631,E2 -3485.631} C_VEL
LIN {X 0,Y 545.111,Z 134.301,A -85,B 0,C 180,E1 -3485.93,E2 -3485.93} C_VEL
LIN {X 0,Y 546.645,Z 142.042,A -85,B 0,C 180,E1 -3487.112,E2 -3487.112} C_VEL
LIN {X 0,Y 546.459,Z 158.317,A -85,B 0,C 180,E1 -3489.406,E2 -3489.406} C_VEL
LIN {X 0,Y 548.463,Z 167.442,A -85,B 0,C 180,E1 -3489.621,E2 -3489.621} C_VEL
LIN {X 0,Y 547.781,Z 322.568,A -85,B 0,C 180,E1 -3491.731,E2 -3491.731} C_VEL
LIN {X 0,Y 547.592,Z 337.926,A -85,B 0,C 180,E1 -3492.083,E2 -3492.083} C_VEL
LIN {X 0,Y 547.303,Z 352.854,A -85,B 0,C 180,E1 -3492.58,E2 -3492.58} C_VEL
LIN {X 0,Y 547.049,Z 366.78,A -85,B 0,C 180,E1 -3493.198,E2 -3493.198} C_VEL
LIN {X 0,Y 546.667,Z 380.347,A -85,B 0,C 180,E1 -3493.953,E2 -3493.953} C_VEL
LIN {X 0,Y 546.289,Z 393.089,A -85,B 0,C 180,E1 -3494.826,E2 -3494.826} C_VEL
LIN {X 0,Y 545.929,Z 405.342,A -85,B 0,C 180,E1 -3495.841,E2 -3495.841} C_VEL
LIN {X 0,Y 545.592,Z 416.715,A -85,B 0,C 180,E1 -3496.971,E2 -3496.971} C_VEL
LIN {X 0,Y 545.266,Z 427.467,A -85,B 0,C 180,E1 -3498.253,E2 -3498.253} C_VEL
LIN {X 0,Y 545.07,Z 436.821,A -85,B 0,C 180,E1 -3499.6,E2 -3499.6} C_VEL
LIN {X 0,Y 544.875,Z 444.439,A -85,B 0,C 180,E1 -3500.908,E2 -3500.908} C_VEL
LIN {X 0,Y 544.819,Z 449.15,A -85,B 0,C 180,E1 -3501.842,E2 -3501.842} C_VEL
LIN {X 0,Y 544.73,Z 453.975,A -85,B 0,C 180,E1 -3502.959,E2 -3502.959} C_VEL
LIN {X 0,Y 544.704,Z 457.998,A -85,B 0,C 180,E1 -3504.075,E2 -3504.075} C_VEL
LIN {X 0,Y 544.605,Z 462.137,A -85,B 0,C 180,E1 -3505.558,E2 -3505.558} C_VEL
LIN {X 0,Y 544.645,Z 463.83,A -85,B 0,C 180,E1 -3506.3,E2 -3506.3} C_VEL
LIN {X 0,Y 544.57,Z 466.122,A -85,B 0,C 180,E1 -3507.78,E2 -3507.78} C_VEL
LIN {X 0,Y 544.537,Z 467.267,A -85,B 0,C 180,E1 -3509.26,E2 -3509.26} C_VEL
LIN {X 0,Y 544.539,Z 467.496,A -85,B 0,C 180,E1 -3509.999,E2 -3509.999} C_VEL
LIN {X 0,Y 544.545,Z 466.943,A -85,B 0,C 180,E1 -3511.478,E2 -3511.478} C_VEL
LIN {X 0,Y 544.645,Z 465.226,A -85,B 0,C 180,E1 -3512.958,E2 -3512.958} C_VEL
LIN {X 0,Y 544.645,Z 464.001,A -85,B 0,C 180,E1 -3513.698,E2 -3513.698} C_VEL
LIN {X 0,Y 544.641,Z 460.531,A -85,B 0,C 180,E1 -3515.181,E2 -3515.181} C_VEL
LIN {X 0,Y 544.697,Z 455.722,A -85,B 0,C 180,E1 -3516.667,E2 -3516.667} C_VEL
LIN {X 0,Y 544.766,Z 451.258,A -85,B 0,C 180,E1 -3517.784,E2 -3517.784} C_VEL
LIN {X 0,Y 544.844,Z 445.93,A -85,B 0,C 180,E1 -3518.904,E2 -3518.904} C_VEL
LIN {X 0,Y 544.975,Z 439.653,A -85,B 0,C 180,E1 -3520.025,E2 -3520.025} C_VEL
LIN {X 0,Y 545.151,Z 432.453,A -85,B 0,C 180,E1 -3521.149,E2 -3521.149} C_VEL
LIN {X 0,Y 545.426,Z 422.458,A -85,B 0,C 180,E1 -3522.463,E2 -3522.463} C_VEL
LIN {X 0,Y 545.713,Z 412.2,A -85,B 0,C 180,E1 -3523.593,E2 -3523.593} C_VEL
LIN {X 0,Y 546.088,Z 399.897,A -85,B 0,C 180,E1 -3524.724,E2 -3524.724} C_VEL
LIN {X 0,Y 546.461,Z 387.494,A -85,B 0,C 180,E1 -3525.668,E2 -3525.668} C_VEL
LIN {X 0,Y 546.877,Z 373.856,A -85,B 0,C 180,E1 -3526.518,E2 -3526.518} C_VEL
LIN {X 0,Y 547.157,Z 359.629,A -85,B 0,C 180,E1 -3527.23,E2 -3527.23} C_VEL
LIN {X 0,Y 547.463,Z 344.805,A -85,B 0,C 180,E1 -3527.799,E2 -3527.799} C_VEL
LIN {X 0,Y 547.688,Z 330.066,A -85,B 0,C 180,E1 -3528.207,E2 -3528.207} C_VEL
LIN {X 0,Y 547.84,Z 313.075,A -85,B 0,C 180,E1 -3528.505,E2 -3528.505} C_VEL
LIN {X 0,Y 548.542,Z 168.455,A -85,B 0,C 180,E1 -3530.453,E2 -3530.453} C_VEL
LIN {X 0,Y 546.473,Z 158.275,A -85,B 0,C 180,E1 -3530.696,E2 -3530.696} C_VEL
LIN {X 0,Y 546.583,Z 141.272,A -85,B 0,C 180,E1 -3533.088,E2 -3533.088} C_VEL
LIN {X 0,Y 545.106,Z 134.211,A -85,B 0,C 180,E1 -3534.203,E2 -3534.203} C_VEL
LIN {X 0,Y 545.09,Z 134.213,A -85,B 0,C 180,E1 -3537.172,E2 -3537.172} C_VEL
LIN {X 0,Y 545.062,Z 134.217,A -85,B 0,C 180,E1 -3539.337,E2 -3539.337} C_VEL
LIN {X 0,Y 545.069,Z 134.211,A -85,B 0,C 180,E1 -3541.912,E2 -3541.912} C_VEL
LIN {X 0,Y 545.08,Z 134.209,A -85,B 0,C 180,E1 -3544.562,E2 -3544.562} C_VEL
LIN {X 0,Y 545.035,Z 134.22,A -85,B 0,C 180,E1 -3547.303,E2 -3547.303} C_VEL
LIN {X 0,Y 545.069,Z 134.204,A -85,B 0,C 180,E1 -3550.141,E2 -3550.141} C_VEL
LIN {X 0,Y 545.08,Z 134.214,A -85,B 0,C 180,E1 -3553.105,E2 -3553.105} C_VEL
LIN {X 0,Y 545.06,Z 134.21,A -85,B 0,C 180,E1 -3556.223,E2 -3556.223} C_VEL
LIN {X 0,Y 545.094,Z 134.209,A -85,B 0,C 180,E1 -3558.886,E2 -3558.886} C_VEL
LIN {X 0,Y 545.047,Z 134.213,A -85,B 0,C 180,E1 -3561.762,E2 -3561.762} C_VEL
LIN {X 0,Y 545.058,Z 134.211,A -85,B 0,C 180,E1 -3564.533,E2 -3564.533} C_VEL
LIN {X 0,Y 545.073,Z 134.217,A -85,B 0,C 180,E1 -3567.212,E2 -3567.212} C_VEL
LIN {X 0,Y 545.093,Z 134.203,A -85,B 0,C 180,E1 -3569.812,E2 -3569.812} C_VEL
LIN {X 0,Y 545.087,Z 134.212,A -85,B 0,C 180,E1 -3572.825,E2 -3572.825} C_VEL
LIN {X 0,Y 545.043,Z 134.211,A -85,B 0,C 180,E1 -3575.63,E2 -3575.63} C_VEL
LIN {X 0,Y 545.06,Z 134.217,A -85,B 0,C 180,E1 -3578.836,E2 -3578.836} C_VEL
LIN {X 0,Y 545.075,Z 134.211,A -85,B 0,C 180,E1 -3581.195,E2 -3581.195} C_VEL
LIN {X 0,Y 545.068,Z 134.211,A -85,B 0,C 180,E1 -3583.521,E2 -3583.521} C_VEL
LIN {X 0,Y 545.086,Z 134.205,A -85,B 0,C 180,E1 -3585.82,E2 -3585.82} C_VEL
LIN {X 0,Y 545.122,Z 134.209,A -85,B 0,C 180,E1 -3588.849,E2 -3588.849} C_VEL
LIN {X 0,Y 545.121,Z 134.201,A -85,B 0,C 180,E1 -3591.847,E2 -3591.847} C_VEL
LIN {X 0,Y 545.199,Z 134.199,A -85,B 0,C 180,E1 -3594.823,E2 -3594.823} C_VEL
LIN {X 0,Y 545.184,Z 134.194,A -85,B 0,C 180,E1 -3597.784,E2 -3597.784} C_VEL
LIN {X 0,Y 545.208,Z 134.195,A -85,B 0,C 180,E1 -3600.739,E2 -3600.739} C_VEL
LIN {X 0,Y 545.167,Z 134.201,A -85,B 0,C 180,E1 -3602.956,E2 -3602.956} C_VEL
LIN {X 0,Y 545.161,Z 134.195,A -85,B 0,C 180,E1 -3605.92,E2 -3605.92} C_VEL
LIN {X 0,Y 545.118,Z 134.206,A -85,B 0,C 180,E1 -3608.9,E2 -3608.9} C_VEL
LIN {X 0,Y 545.125,Z 134.201,A -85,B 0,C 180,E1 -3611.904,E2 -3611.904} C_VEL
LIN {X 0,Y 545.075,Z 134.21,A -85,B 0,C 180,E1 -3614.944,E2 -3614.944} C_VEL
LIN {X 0,Y 545.073,Z 134.21,A -85,B 0,C 180,E1 -3618.026,E2 -3618.026} C_VEL
LIN {X 0,Y 545.089,Z 134.211,A -85,B 0,C 180,E1 -3620.372,E2 -3620.372} C_VEL
LIN {X 0,Y 545.104,Z 134.203,A -85,B 0,C 180,E1 -3623.558,E2 -3623.558} C_VEL
LIN {X 0,Y 545.07,Z 134.211,A -85,B 0,C 180,E1 -3626.001,E2 -3626.001} C_VEL
LIN {X 0,Y 545.081,Z 134.207,A -85,B 0,C 180,E1 -3628.749,E2 -3628.749} C_VEL
LIN {X 0,Y 545.068,Z 134.21,A -85,B 0,C 180,E1 -3631.683,E2 -3631.683} C_VEL
LIN {X 0,Y 545.072,Z 134.212,A -85,B 0,C 180,E1 -3634.564,E2 -3634.564} C_VEL
LIN {X 0,Y 545.03,Z 134.213,A -85,B 0,C 180,E1 -3637.304,E2 -3637.304} C_VEL
LIN {X 0,Y 545.064,Z 134.207,A -85,B 0,C 180,E1 -3640.143,E2 -3640.143} C_VEL
LIN {X 0,Y 545.054,Z 134.212,A -85,B 0,C 180,E1 -3642.698,E2 -3642.698} C_VEL
LIN {X 0,Y 545.055,Z 134.211,A -85,B 0,C 180,E1 -3645.168,E2 -3645.168} C_VEL
LIN {X 0,Y 545.076,Z 134.216,A -85,B 0,C 180,E1 -3647.899,E2 -3647.899} C_VEL
LIN {X 0,Y 545.098,Z 134.206,A -85,B 0,C 180,E1 -3650.677,E2 -3650.677} C_VEL
LIN {X 0,Y 545.047,Z 134.215,A -85,B 0,C 180,E1 -3653.622,E2 -3653.622} C_VEL
LIN {X 0,Y 545.063,Z 134.213,A -85,B 0,C 180,E1 -3656.329,E2 -3656.329} C_VEL
LIN {X 0,Y 545.062,Z 134.213,A -85,B 0,C 180,E1 -3658.953,E2 -3658.953} C_VEL
LIN {X 0,Y 545.095,Z 134.319,A -85,B 0,C 180,E1 -3659.934,E2 -3659.934} C_VEL
LIN {X 0,Y 548.994,Z 147.48,A -85,B 0,C 180,E1 -3661.338,E2 -3661.338} C_VEL
LIN {X 0,Y 548.418,Z 173.897,A -85,B 0,C 180,E1 -3663.645,E2 -3663.645} C_VEL
LIN {X 0,Y 547.612,Z 210.439,A -85,B 0,C 180,E1 -3666.758,E2 -3666.758} C_VEL
LIN {X 0,Y 547.029,Z 242.727,A -85,B 0,C 180,E1 -3669.434,E2 -3669.434} C_VEL
LIN {X 0,Y 548.255,Z 253.227,A -85,B 0,C 180,E1 -3669.621,E2 -3669.621} C_VEL
LIN {X 0,Y 547.6,Z 411.715,A -85,B 0,C 180,E1 -3671.745,E2 -3671.745} C_VEL
LIN {X 0,Y 547.397,Z 427.184,A -85,B 0,C 180,E1 -3672.103,E2 -3672.103} C_VEL
LIN {X 0,Y 547.129,Z 442.783,A -85,B 0,C 180,E1 -3672.625,E2 -3672.625} C_VEL
LIN {X 0,Y 546.821,Z 455.797,A -85,B 0,C 180,E1 -3673.192,E2 -3673.192} C_VEL
LIN {X 0,Y 546.522,Z 469.737,A -85,B 0,C 180,E1 -3673.951,E2 -3673.951} C_VEL
LIN {X 0,Y 546.217,Z 482.448,A -85,B 0,C 180,E1 -3674.796,E2 -3674.796} C_VEL
LIN {X 0,Y 545.87,Z 494.229,A -85,B 0,C 180,E1 -3675.746,E2 -3675.746} C_VEL
LIN {X 0,Y 545.588,Z 504.975,A -85,B 0,C 180,E1 -3676.784,E2 -3676.784} C_VEL
LIN {X 0,Y 545.314,Z 514.913,A -85,B 0,C 180,E1 -3677.912,E2 -3677.912} C_VEL
LIN {X 0,Y 545.135,Z 524.63,A -85,B 0,C 180,E1 -3679.227,E2 -3679.227} C_VEL
LIN {X 0,Y 544.89,Z 532.733,A -85,B 0,C 180,E1 -3680.536,E2 -3680.536} C_VEL
LIN {X 0,Y 544.817,Z 539.427,A -85,B 0,C 180,E1 -3681.843,E2 -3681.843} C_VEL
LIN {X 0,Y 544.703,Z 546.083,A -85,B 0,C 180,E1 -3683.457,E2 -3683.457} C_VEL
LIN {X 0,Y 544.642,Z 550.388,A -85,B 0,C 180,E1 -3684.819,E2 -3684.819} C_VEL
LIN {X 0,Y 544.644,Z 553.889,A -85,B 0,C 180,E1 -3686.302,E2 -3686.302} C_VEL
LIN {X 0,Y 544.569,Z 556.191,A -85,B 0,C 180,E1 -3687.782,E2 -3687.782} C_VEL
LIN {X 0,Y 544.539,Z 557.348,A -85,B 0,C 180,E1 -3689.261,E2 -3689.261} C_VEL
LIN {X 0,Y 544.539,Z 557.347,A -85,B 0,C 180,E1 -3690.74,E2 -3690.74} C_VEL
LIN {X 0,Y 544.57,Z 556.185,A -85,B 0,C 180,E1 -3692.22,E2 -3692.22} C_VEL
LIN {X 0,Y 544.644,Z 553.881,A -85,B 0,C 180,E1 -3693.7,E2 -3693.7} C_VEL
LIN {X 0,Y 544.642,Z 550.384,A -85,B 0,C 180,E1 -3695.183,E2 -3695.183} C_VEL
LIN {X 0,Y 544.698,Z 545.606,A -85,B 0,C 180,E1 -3696.669,E2 -3696.669} C_VEL
LIN {X 0,Y 544.819,Z 539.416,A -85,B 0,C 180,E1 -3698.158,E2 -3698.158} C_VEL
LIN {X 0,Y 544.905,Z 531.638,A -85,B 0,C 180,E1 -3699.653,E2 -3699.653} C_VEL
LIN {X 0,Y 545.151,Z 523.361,A -85,B 0,C 180,E1 -3700.963,E2 -3700.963} C_VEL
LIN {X 0,Y 545.359,Z 513.384,A -85,B 0,C 180,E1 -3702.278,E2 -3702.278} C_VEL
LIN {X 0,Y 545.64,Z 503.174,A -85,B 0,C 180,E1 -3703.407,E2 -3703.407} C_VEL
LIN {X 0,Y 545.976,Z 490.995,A -85,B 0,C 180,E1 -3704.538,E2 -3704.538} C_VEL
LIN {X 0,Y 546.349,Z 478.384,A -85,B 0,C 180,E1 -3705.494,E2 -3705.494} C_VEL
LIN {X 0,Y 546.626,Z 464.734,A -85,B 0,C 180,E1 -3706.336,E2 -3706.336} C_VEL
LIN {X 0,Y 546.936,Z 449.407,A -85,B 0,C 180,E1 -3707.095,E2 -3707.095} C_VEL
LIN {X 0,Y 547.216,Z 433.714,A -85,B 0,C 180,E1 -3707.688,E2 -3707.688} C_VEL
LIN {X 0,Y 547.454,Z 418.567,A -85,B 0,C 180,E1 -3708.103,E2 -3708.103} C_VEL
LIN {X 0,Y 547.597,Z 402.305,A -85,B 0,C 180,E1 -3708.386,E2 -3708.386} C_VEL
LIN {X 0,Y 548.218,Z 251.727,A -85,B 0,C 180,E1 -3710.384,E2 -3710.384} C_VEL
LIN {X 0,Y 546.959,Z 242.397,A -85,B 0,C 180,E1 -3710.557,E2 -3710.557} C_VEL
LIN {X 0,Y 547.549,Z 206.009,A -85,B 0,C 180,E1 -3713.548,E2 -3713.548} C_VEL
LIN {X 0,Y 548.325,Z 169.455,A -85,B 0,C 180,E1 -3716.655,E2 -3716.655} C_VEL
LIN {X 0,Y 548.846,Z 147.843,A -85,B 0,C 180,E1 -3718.563,E2 -3718.563} C_VEL
LIN {X 0,Y 546.533,Z 139.149,A -85,B 0,C 180,E1 -3719.491,E2 -3719.491} C_VEL
LIN {X 0,Y 545.056,Z 134.219,A -85,B 0,C 180,E1 -3720.057,E2 -3720.057} C_VEL
LIN {X 0,Y 545.08,Z 134.213,A -85,B 0,C 180,E1 -3723.062,E2 -3723.062} C_VEL
LIN {X 0,Y 545.024,Z 134.224,A -85,B 0,C 180,E1 -3725.671,E2 -3725.671} C_VEL
LIN {X 0,Y 545.047,Z 134.216,A -85,B 0,C 180,E1 -3728.239,E2 -3728.239} C_VEL
LIN {X 0,Y 545.013,Z 134.221,A -85,B 0,C 180,E1 -3731.122,E2 -3731.122} C_VEL
LIN {X 0,Y 545.027,Z 134.217,A -85,B 0,C 180,E1 -3734.133,E2 -3734.133} C_VEL
LIN {X 0,Y 545.018,Z 134.22,A -85,B 0,C 180,E1 -3736.888,E2 -3736.888} C_VEL
LIN {X 0,Y 545.007,Z 134.22,A -85,B 0,C 180,E1 -3739.852,E2 -3739.852} C_VEL
LIN {X 0,Y 545.006,Z 134.223,A -85,B 0,C 180,E1 -3742.694,E2 -3742.694} C_VEL
LIN {X 0,Y 545.055,Z 134.214,A -85,B 0,C 180,E1 -3745.612,E2 -3745.612} C_VEL
LIN {X 0,Y 545.046,Z 134.217,A -85,B 0,C 180,E1 -3748.324,E2 -3748.324} C_VEL
LIN {X 0,Y 545.042,Z 134.217,A -85,B 0,C 180,E1 -3751.504,E2 -3751.504} C_VEL
LIN {X 0,Y 545.048,Z 134.22,A -85,B 0,C 180,E1 -3753.998,E2 -3753.998} C_VEL
LIN {X 0,Y 545.067,Z 134.305,A -85,B 0,C 180,E1 -3755.403,E2 -3755.403} C_VEL
LIN {X 0,Y 547.083,Z 142.993,A -85,B 0,C 180,E1 -3756.933,E2 -3756.933} C_VEL
LIN {X 0,Y 546.865,Z 155.505,A -85,B 0,C 180,E1 -3758.91,E2 -3758.91} C_VEL
LIN {X 0,Y 546.337,Z 174.221,A -85,B 0,C 180,E1 -3761.823,E2 -3761.823} C_VEL
LIN {X 0,Y 545.836,Z 193.062,A -85,B 0,C 180,E1 -3764.734,E2 -3764.734} C_VEL
LIN {X 0,Y 545.794,Z 196.987,A -85,B 0,C 180,E1 -3765.335,E2 -3765.335} C_VEL
LIN {X 0,Y 546.845,Z 202.478,A -85,B 0,C 180,E1 -3765.464,E2 -3765.464} C_VEL
LIN {X 0,Y 546.279,Z 307.287,A -85,B 0,C 180,E1 -3766.989,E2 -3766.989} C_VEL
LIN {X 0,Y 546.166,Z 320.571,A -85,B 0,C 180,E1 -3767.341,E2 -3767.341} C_VEL
LIN {X 0,Y 546.042,Z 333.39,A -85,B 0,C 180,E1 -3767.843,E2 -3767.843} C_VEL
LIN {X 0,Y 545.818,Z 345.788,A -85,B 0,C 180,E1 -3768.502,E2 -3768.502} C_VEL
LIN {X 0,Y 545.632,Z 356.583,A -85,B 0,C 180,E1 -3769.236,E2 -3769.236} C_VEL
LIN {X 0,Y 545.435,Z 365.497,A -85,B 0,C 180,E1 -3769.983,E2 -3769.983} C_VEL
LIN {X 0,Y 545.255,Z 374.632,A -85,B 0,C 180,E1 -3770.915,E2 -3770.915} C_VEL
LIN {X 0,Y 545.058,Z 383.455,A -85,B 0,C 180,E1 -3772.033,E2 -3772.033} C_VEL
LIN {X 0,Y 544.926,Z 391.171,A -85,B 0,C 180,E1 -3773.259,E2 -3773.259} C_VEL
LIN {X 0,Y 544.829,Z 396.996,A -85,B 0,C 180,E1 -3774.448,E2 -3774.448} C_VEL
LIN {X 0,Y 544.789,Z 401.245,A -85,B 0,C 180,E1 -3775.561,E2 -3775.561} C_VEL
LIN {X 0,Y 544.739,Z 403.489,A -85,B 0,C 180,E1 -3776.301,E2 -3776.301} C_VEL
LIN {X 0,Y 544.706,Z 405.312,A -85,B 0,C 180,E1 -3777.042,E2 -3777.042} C_VEL
LIN {X 0,Y 544.651,Z 406.696,A -85,B 0,C 180,E1 -3777.782,E2 -3777.782} C_VEL
LIN {X 0,Y 544.635,Z 408.268,A -85,B 0,C 180,E1 -3779.261,E2 -3779.261} C_VEL
LIN {X 0,Y 544.63,Z 408.485,A -85,B 0,C 180,E1 -3780,E2 -3780} C_VEL
LIN {X 0,Y 544.634,Z 408.297,A -85,B 0,C 180,E1 -3780.739,E2 -3780.739} C_VEL
LIN {X 0,Y 544.65,Z 406.764,A -85,B 0,C 180,E1 -3782.219,E2 -3782.219} C_VEL
LIN {X 0,Y 544.696,Z 405.405,A -85,B 0,C 180,E1 -3782.958,E2 -3782.958} C_VEL
LIN {X 0,Y 544.76,Z 402.561,A -85,B 0,C 180,E1 -3784.069,E2 -3784.069} C_VEL
LIN {X 0,Y 544.708,Z 398.724,A -85,B 0,C 180,E1 -3785.182,E2 -3785.182} C_VEL
LIN {X 0,Y 544.866,Z 393.347,A -85,B 0,C 180,E1 -3786.373,E2 -3786.373} C_VEL
LIN {X 0,Y 544.952,Z 386.265,A -85,B 0,C 180,E1 -3787.596,E2 -3787.596} C_VEL
LIN {X 0,Y 545.123,Z 378.14,A -85,B 0,C 180,E1 -3788.713,E2 -3788.713} C_VEL
LIN {X 0,Y 545.299,Z 369.802,A -85,B 0,C 180,E1 -3789.645,E2 -3789.645} C_VEL
LIN {X 0,Y 545.532,Z 359.491,A -85,B 0,C 180,E1 -3790.578,E2 -3790.578} C_VEL
LIN {X 0,Y 545.716,Z 347.824,A -85,B 0,C 180,E1 -3791.422,E2 -3791.422} C_VEL
LIN {X 0,Y 545.922,Z 336.238,A -85,B 0,C 180,E1 -3792.075,E2 -3792.075} C_VEL
LIN {X 0,Y 545.989,Z 324.16,A -85,B 0,C 180,E1 -3792.593,E2 -3792.593} C_VEL
LIN {X 0,Y 546.19,Z 311.033,A -85,B 0,C 180,E1 -3792.99,E2 -3792.99} C_VEL
LIN {X 0,Y 546.291,Z 298.478,A -85,B 0,C 180,E1 -3793.224,E2 -3793.224} C_VEL
LIN {X 0,Y 546.54,Z 201.943,A -85,B 0,C 180,E1 -3794.539,E2 -3794.539} C_VEL
LIN {X 0,Y 545.519,Z 195.963,A -85,B 0,C 180,E1 -3794.678,E2 -3794.678} C_VEL
LIN {X 0,Y 545.858,Z 175.514,A -85,B 0,C 180,E1 -3797.762,E2 -3797.762} C_VEL
LIN {X 0,Y 546.27,Z 157.315,A -85,B 0,C 180,E1 -3800.523,E2 -3800.523} C_VEL
LIN {X 0,Y 546.372,Z 150.344,A -85,B 0,C 180,E1 -3801.595,E2 -3801.595} C_VEL
LIN {X 0,Y 545.781,Z 148.259,A -85,B 0,C 180,E1 -3801.941,E2 -3801.941} C_VEL
LIN {X 0,Y 543.124,Z 145.371,A -85,B 0,C 180,E1 -3802.51,E2 -3802.51} C_VEL
LIN {X 0,Y 539.762,Z 141.948,A -85,B 0,C 180,E1 -3803.205,E2 -3803.205} C_VEL
LIN {X 0,Y 539.202,Z 140.592,A -85,B 0,C 180,E1 -3803.445,E2 -3803.445} C_VEL
LIN {X 0,Y 538.037,Z 135.091,A -85,B 0,C 180,E1 -3804.399,E2 -3804.399} C_VEL
LIN {X 0,Y 538.019,Z 135.095,A -85,B 0,C 180,E1 -3807.206,E2 -3807.206} C_VEL
LIN {X 0,Y 538.016,Z 135.093,A -85,B 0,C 180,E1 -3809.761,E2 -3809.761} C_VEL
LIN {X 0,Y 538.022,Z 135.088,A -85,B 0,C 180,E1 -3812.383,E2 -3812.383} C_VEL
LIN {X 0,Y 537.999,Z 135.096,A -85,B 0,C 180,E1 -3815.084,E2 -3815.084} C_VEL
LIN {X 0,Y 537.993,Z 135.092,A -85,B 0,C 180,E1 -3817.878,E2 -3817.878} C_VEL
LIN {X 0,Y 538.026,Z 135.087,A -85,B 0,C 180,E1 -3820.778,E2 -3820.778} C_VEL
LIN {X 0,Y 538.024,Z 135.085,A -85,B 0,C 180,E1 -3824.073,E2 -3824.073} C_VEL
LIN {X 0,Y 538.024,Z 135.093,A -85,B 0,C 180,E1 -3827.214,E2 -3827.214} C_VEL
LIN {X 0,Y 538.015,Z 135.087,A -85,B 0,C 180,E1 -3830.202,E2 -3830.202} C_VEL
LIN {X 0,Y 538.029,Z 135.094,A -85,B 0,C 180,E1 -3833.067,E2 -3833.067} C_VEL
LIN {X 0,Y 538.014,Z 135.09,A -85,B 0,C 180,E1 -3835.826,E2 -3835.826} C_VEL
LIN {X 0,Y 538.013,Z 135.096,A -85,B 0,C 180,E1 -3838.498,E2 -3838.498} C_VEL
LIN {X 0,Y 538.024,Z 135.092,A -85,B 0,C 180,E1 -3841.097,E2 -3841.097} C_VEL
LIN {X 0,Y 538.045,Z 135.087,A -85,B 0,C 180,E1 -3843.633,E2 -3843.633} C_VEL
LIN {X 0,Y 538.067,Z 135.219,A -85,B 0,C 180,E1 -3845.704,E2 -3845.704} C_VEL
LIN {X 0,Y 539.785,Z 143.622,A -85,B 0,C 180,E1 -3847.007,E2 -3847.007} C_VEL
LIN {X 0,Y 539.63,Z 158.699,A -85,B 0,C 180,E1 -3849.13,E2 -3849.13} C_VEL
LIN {X 0,Y 541.902,Z 169.301,A -85,B 0,C 180,E1 -3849.382,E2 -3849.382} C_VEL
LIN {X 0,Y 541.069,Z 323.866,A -85,B 0,C 180,E1 -3851.511,E2 -3851.511} C_VEL
LIN {X 0,Y 540.884,Z 339.307,A -85,B 0,C 180,E1 -3851.878,E2 -3851.878} C_VEL
LIN {X 0,Y 540.565,Z 353.408,A -85,B 0,C 180,E1 -3852.356,E2 -3852.356} C_VEL
LIN {X 0,Y 540.283,Z 367.344,A -85,B 0,C 180,E1 -3852.981,E2 -3852.981} C_VEL
LIN {X 0,Y 539.876,Z 380.918,A -85,B 0,C 180,E1 -3853.746,E2 -3853.746} C_VEL
LIN {X 0,Y 539.42,Z 394.499,A -85,B 0,C 180,E1 -3854.693,E2 -3854.693} C_VEL
LIN {X 0,Y 539.037,Z 406.95,A -85,B 0,C 180,E1 -3855.753,E2 -3855.753} C_VEL
LIN {X 0,Y 538.694,Z 417.297,A -85,B 0,C 180,E1 -3856.801,E2 -3856.801} C_VEL
LIN {X 0,Y 538.316,Z 428.201,A -85,B 0,C 180,E1 -3858.12,E2 -3858.12} C_VEL
LIN {X 0,Y 538.086,Z 437.4,A -85,B 0,C 180,E1 -3859.463,E2 -3859.463} C_VEL
LIN {X 0,Y 537.88,Z 444,A -85,B 0,C 180,E1 -3860.599,E2 -3860.599} C_VEL
LIN {X 0,Y 537.724,Z 451.239,A -85,B 0,C 180,E1 -3862.111,E2 -3862.111} C_VEL
LIN {X 0,Y 537.619,Z 456.471,A -85,B 0,C 180,E1 -3863.468,E2 -3863.468} C_VEL
LIN {X 0,Y 537.574,Z 460.376,A -85,B 0,C 180,E1 -3864.748,E2 -3864.748} C_VEL
LIN {X 0,Y 537.562,Z 463.847,A -85,B 0,C 180,E1 -3866.251,E2 -3866.251} C_VEL
LIN {X 0,Y 537.488,Z 466.116,A -85,B 0,C 180,E1 -3867.751,E2 -3867.751} C_VEL
LIN {X 0,Y 537.437,Z 467.259,A -85,B 0,C 180,E1 -3869.25,E2 -3869.25} C_VEL
LIN {X 0,Y 537.44,Z 467.496,A -85,B 0,C 180,E1 -3869.999,E2 -3869.999} C_VEL
LIN {X 0,Y 537.45,Z 466.936,A -85,B 0,C 180,E1 -3871.498,E2 -3871.498} C_VEL
LIN {X 0,Y 537.545,Z 465.228,A -85,B 0,C 180,E1 -3872.997,E2 -3872.997} C_VEL
LIN {X 0,Y 537.509,Z 462.441,A -85,B 0,C 180,E1 -3874.499,E2 -3874.499} C_VEL
LIN {X 0,Y 537.617,Z 458.475,A -85,B 0,C 180,E1 -3876.002,E2 -3876.002} C_VEL
LIN {X 0,Y 537.674,Z 453.168,A -85,B 0,C 180,E1 -3877.51,E2 -3877.51} C_VEL
LIN {X 0,Y 537.841,Z 446.404,A -85,B 0,C 180,E1 -3879.02,E2 -3879.02} C_VEL
LIN {X 0,Y 538.071,Z 439.154,A -85,B 0,C 180,E1 -3880.345,E2 -3880.345} C_VEL
LIN {X 0,Y 538.28,Z 430.249,A -85,B 0,C 180,E1 -3881.697,E2 -3881.697} C_VEL
LIN {X 0,Y 538.613,Z 419.836,A -85,B 0,C 180,E1 -3883.007,E2 -3883.007} C_VEL
LIN {X 0,Y 538.978,Z 408.967,A -85,B 0,C 180,E1 -3884.151,E2 -3884.151} C_VEL
LIN {X 0,Y 539.396,Z 396.672,A -85,B 0,C 180,E1 -3885.228,E2 -3885.228} C_VEL
LIN {X 0,Y 539.771,Z 383.867,A -85,B 0,C 180,E1 -3886.158,E2 -3886.158} C_VEL
LIN {X 0,Y 540.209,Z 371.007,A -85,B 0,C 180,E1 -3886.922,E2 -3886.922} C_VEL
LIN {X 0,Y 540.493,Z 356.935,A -85,B 0,C 180,E1 -3887.596,E2 -3887.596} C_VEL
LIN {X 0,Y 540.836,Z 341.66,A -85,B 0,C 180,E1 -3888.146,E2 -3888.146} C_VEL
LIN {X 0,Y 541.023,Z 326.807,A -85,B 0,C 180,E1 -3888.526,E2 -3888.526} C_VEL
LIN {X 0,Y 541.153,Z 303.27,A -85,B 0,C 180,E1 -3888.882,E2 -3888.882} C_VEL
LIN {X 0,Y 541.927,Z 168.959,A -85,B 0,C 180,E1 -3890.713,E2 -3890.713} C_VEL
LIN {X 0,Y 539.675,Z 158.63,A -85,B 0,C 180,E1 -3890.969,E2 -3890.969} C_VEL
LIN {X 0,Y 539.849,Z 144.243,A -85,B 0,C 180,E1 -3892.988,E2 -3892.988} C_VEL
LIN {X 0,Y 538.052,Z 135.089,A -85,B 0,C 180,E1 -3894.426,E2 -3894.426} C_VEL
LIN {X 0,Y 538.055,Z 135.091,A -85,B 0,C 180,E1 -3897.351,E2 -3897.351} C_VEL
LIN {X 0,Y 538.015,Z 135.096,A -85,B 0,C 180,E1 -3899.76,E2 -3899.76} C_VEL
LIN {X 0,Y 538.029,Z 135.085,A -85,B 0,C 180,E1 -3902.381,E2 -3902.381} C_VEL
LIN {X 0,Y 538.017,Z 135.093,A -85,B 0,C 180,E1 -3905.081,E2 -3905.081} C_VEL
LIN {X 0,Y 537.989,Z 135.094,A -85,B 0,C 180,E1 -3907.876,E2 -3907.876} C_VEL
LIN {X 0,Y 538.046,Z 135.079,A -85,B 0,C 180,E1 -3910.774,E2 -3910.774} C_VEL
LIN {X 0,Y 538.022,Z 135.085,A -85,B 0,C 180,E1 -3914.074,E2 -3914.074} C_VEL
LIN {X 0,Y 538.019,Z 135.093,A -85,B 0,C 180,E1 -3917.011,E2 -3917.011} C_VEL
LIN {X 0,Y 538.071,Z 135.09,A -85,B 0,C 180,E1 -3919.248,E2 -3919.248} C_VEL
LIN {X 0,Y 537.986,Z 135.091,A -85,B 0,C 180,E1 -3922.122,E2 -3922.122} C_VEL
LIN {X 0,Y 538.013,Z 135.093,A -85,B 0,C 180,E1 -3924.917,E2 -3924.917} C_VEL
LIN {X 0,Y 538.023,Z 135.089,A -85,B 0,C 180,E1 -3927.617,E2 -3927.617} C_VEL
LIN {X 0,Y 538.034,Z 135.081,A -85,B 0,C 180,E1 -3930.24,E2 -3930.24} C_VEL
LIN {X 0,Y 538.057,Z 135.088,A -85,B 0,C 180,E1 -3932.796,E2 -3932.796} C_VEL
LIN {X 0,Y 538.039,Z 135.087,A -85,B 0,C 180,E1 -3935.292,E2 -3935.292} C_VEL
LIN {X 0,Y 538.005,Z 135.089,A -85,B 0,C 180,E1 -3938.041,E2 -3938.041} C_VEL
LIN {X 0,Y 538.031,Z 135.089,A -85,B 0,C 180,E1 -3940.94,E2 -3940.94} C_VEL
LIN {X 0,Y 538.018,Z 135.091,A -85,B 0,C 180,E1 -3943.299,E2 -3943.299} C_VEL
LIN {X 0,Y 538.054,Z 135.081,A -85,B 0,C 180,E1 -3945.63,E2 -3945.63} C_VEL
LIN {X 0,Y 538.079,Z 135.083,A -85,B 0,C 180,E1 -3948.701,E2 -3948.701} C_VEL
LIN {X 0,Y 538.078,Z 135.078,A -85,B 0,C 180,E1 -3951.739,E2 -3951.739} C_VEL
LIN {X 0,Y 538.156,Z 135.074,A -85,B 0,C 180,E1 -3954.755,E2 -3954.755} C_VEL
LIN {X 0,Y 538.156,Z 135.07,A -85,B 0,C 180,E1 -3957.755,E2 -3957.755} C_VEL
LIN {X 0,Y 538.177,Z 135.071,A -85,B 0,C 180,E1 -3960.748,E2 -3960.748} C_VEL
LIN {X 0,Y 538.133,Z 135.077,A -85,B 0,C 180,E1 -3962.994,E2 -3962.994} C_VEL
LIN {X 0,Y 538.114,Z 135.073,A -85,B 0,C 180,E1 -3965.997,E2 -3965.997} C_VEL
LIN {X 0,Y 538.067,Z 135.083,A -85,B 0,C 180,E1 -3969.018,E2 -3969.018} C_VEL
LIN {X 0,Y 538.073,Z 135.08,A -85,B 0,C 180,E1 -3972.063,E2 -3972.063} C_VEL
LIN {X 0,Y 538.035,Z 135.085,A -85,B 0,C 180,E1 -3975.144,E2 -3975.144} C_VEL
LIN {X 0,Y 538.025,Z 135.091,A -85,B 0,C 180,E1 -3978.27,E2 -3978.27} C_VEL
LIN {X 0,Y 538.032,Z 135.09,A -85,B 0,C 180,E1 -3980.652,E2 -3980.652} C_VEL
LIN {X 0,Y 538.031,Z 135.086,A -85,B 0,C 180,E1 -3983.887,E2 -3983.887} C_VEL
LIN {X 0,Y 538.033,Z 135.093,A -85,B 0,C 180,E1 -3986.367,E2 -3986.367} C_VEL
LIN {X 0,Y 538.022,Z 135.085,A -85,B 0,C 180,E1 -3988.934,E2 -3988.934} C_VEL
LIN {X 0,Y 538.018,Z 135.091,A -85,B 0,C 180,E1 -3991.891,E2 -3991.891} C_VEL
LIN {X 0,Y 538.022,Z 135.089,A -85,B 0,C 180,E1 -3994.622,E2 -3994.622} C_VEL
LIN {X 0,Y 537.999,Z 135.089,A -85,B 0,C 180,E1 -3997.171,E2 -3997.171} C_VEL
LIN {X 0,Y 538.019,Z 135.085,A -85,B 0,C 180,E1 -3999.797,E2 -3999.797} C_VEL
LIN {X 0,Y 538.01,Z 135.089,A -85,B 0,C 180,E1 -4002.787,E2 -4002.787} C_VEL
LIN {X 0,Y 538.024,Z 135.087,A -85,B 0,C 180,E1 -4005.142,E2 -4005.142} C_VEL
LIN {X 0,Y 538.034,Z 135.092,A -85,B 0,C 180,E1 -4008.229,E2 -4008.229} C_VEL
LIN {X 0,Y 538.052,Z 135.086,A -85,B 0,C 180,E1 -4010.413,E2 -4010.413} C_VEL
LIN {X 0,Y 538.022,Z 135.086,A -85,B 0,C 180,E1 -4013.069,E2 -4013.069} C_VEL
LIN {X 0,Y 538.019,Z 135.092,A -85,B 0,C 180,E1 -4015.828,E2 -4015.828} C_VEL
LIN {X 0,Y 538.005,Z 135.094,A -85,B 0,C 180,E1 -4018.5,E2 -4018.5} C_VEL
LIN {X 0,Y 538.034,Z 135.143,A -85,B 0,C 180,E1 -4019.612,E2 -4019.612} C_VEL
LIN {X 0,Y 542.374,Z 149.754,A -85,B 0,C 180,E1 -4021.197,E2 -4021.197} C_VEL
LIN {X 0,Y 541.654,Z 176.283,A -85,B 0,C 180,E1 -4023.544,E2 -4023.544} C_VEL
LIN {X 0,Y 540.801,Z 211.051,A -85,B 0,C 180,E1 -4026.549,E2 -4026.549} C_VEL
LIN {X 0,Y 540.135,Z 242.459,A -85,B 0,C 180,E1 -4029.197,E2 -4029.197} C_VEL
LIN {X 0,Y 541.496,Z 253.708,A -85,B 0,C 180,E1 -4029.406,E2 -4029.406} C_VEL
LIN {X 0,Y 540.714,Z 410.639,A -85,B 0,C 180,E1 -4031.542,E2 -4031.542} C_VEL
LIN {X 0,Y 540.475,Z 426.648,A -85,B 0,C 180,E1 -4031.914,E2 -4031.914} C_VEL
LIN {X 0,Y 540.209,Z 442.204,A -85,B 0,C 180,E1 -4032.444,E2 -4032.444} C_VEL
LIN {X 0,Y 539.848,Z 456.189,A -85,B 0,C 180,E1 -4033.066,E2 -4033.066} C_VEL
LIN {X 0,Y 539.512,Z 469.909,A -85,B 0,C 180,E1 -4033.834,E2 -4033.834} C_VEL
LIN {X 0,Y 539.129,Z 483.842,A -85,B 0,C 180,E1 -4034.791,E2 -4034.791} C_VEL
LIN {X 0,Y 538.767,Z 496.503,A -85,B 0,C 180,E1 -4035.844,E2 -4035.844} C_VEL
LIN {X 0,Y 538.486,Z 508.041,A -85,B 0,C 180,E1 -4036.99,E2 -4036.99} C_VEL
LIN {X 0,Y 538.177,Z 518.61,A -85,B 0,C 180,E1 -4038.243,E2 -4038.243} C_VEL
LIN {X 0,Y 538.023,Z 527.088,A -85,B 0,C 180,E1 -4039.464,E2 -4039.464} C_VEL
LIN {X 0,Y 537.796,Z 535.753,A -85,B 0,C 180,E1 -4040.979,E2 -4040.979} C_VEL
LIN {X 0,Y 537.66,Z 542.703,A -85,B 0,C 180,E1 -4042.49,E2 -4042.49} C_VEL
LIN {X 0,Y 537.623,Z 548.164,A -85,B 0,C 180,E1 -4043.998,E2 -4043.998} C_VEL
LIN {X 0,Y 537.507,Z 552.292,A -85,B 0,C 180,E1 -4045.501,E2 -4045.501} C_VEL
LIN {X 0,Y 537.544,Z 555.185,A -85,B 0,C 180,E1 -4047.003,E2 -4047.003} C_VEL
LIN {X 0,Y 537.449,Z 556.91,A -85,B 0,C 180,E1 -4048.502,E2 -4048.502} C_VEL
LIN {X 0,Y 537.439,Z 557.5,A -85,B 0,C 180,E1 -4050.001,E2 -4050.001} C_VEL
LIN {X 0,Y 537.449,Z 556.906,A -85,B 0,C 180,E1 -4051.5,E2 -4051.5} C_VEL
LIN {X 0,Y 537.544,Z 555.177,A -85,B 0,C 180,E1 -4052.999,E2 -4052.999} C_VEL
LIN {X 0,Y 537.507,Z 552.286,A -85,B 0,C 180,E1 -4054.5,E2 -4054.5} C_VEL
LIN {X 0,Y 537.62,Z 548.162,A -85,B 0,C 180,E1 -4056.004,E2 -4056.004} C_VEL
LIN {X 0,Y 537.662,Z 542.697,A -85,B 0,C 180,E1 -4057.512,E2 -4057.512} C_VEL
LIN {X 0,Y 537.798,Z 535.738,A -85,B 0,C 180,E1 -4059.023,E2 -4059.023} C_VEL
LIN {X 0,Y 538.025,Z 527.074,A -85,B 0,C 180,E1 -4060.538,E2 -4060.538} C_VEL
LIN {X 0,Y 538.192,Z 518.539,A -85,B 0,C 180,E1 -4061.766,E2 -4061.766} C_VEL
LIN {X 0,Y 538.486,Z 507.981,A -85,B 0,C 180,E1 -4063.012,E2 -4063.012} C_VEL
LIN {X 0,Y 538.78,Z 496.362,A -85,B 0,C 180,E1 -4064.158,E2 -4064.158} C_VEL
LIN {X 0,Y 539.13,Z 484.183,A -85,B 0,C 180,E1 -4065.165,E2 -4065.165} C_VEL
LIN {X 0,Y 539.457,Z 471.015,A -85,B 0,C 180,E1 -4066.073,E2 -4066.073} C_VEL
LIN {X 0,Y 539.798,Z 457.451,A -85,B 0,C 180,E1 -4066.84,E2 -4066.84} C_VEL
LIN {X 0,Y 540.09,Z 443.751,A -85,B 0,C 180,E1 -4067.465,E2 -4067.465} C_VEL
LIN {X 0,Y 540.401,Z 428.727,A -85,B 0,C 180,E1 -4067.992,E2 -4067.992} C_VEL
LIN {X 0,Y 540.573,Z 413.916,A -85,B 0,C 180,E1 -4068.364,E2 -4068.364} C_VEL
LIN {X 0,Y 540.71,Z 391.64,A -85,B 0,C 180,E1 -4068.703,E2 -4068.703} C_VEL
LIN {X 0,Y 541.378,Z 252.107,A -85,B 0,C 180,E1 -4070.594,E2 -4070.594} C_VEL
LIN {X 0,Y 540.044,Z 241.868,A -85,B 0,C 180,E1 -4070.796,E2 -4070.796} C_VEL
LIN {X 0,Y 540.707,Z 207.6,A -85,B 0,C 180,E1 -4073.661,E2 -4073.661} C_VEL
LIN {X 0,Y 541.563,Z 172.085,A -85,B 0,C 180,E1 -4076.729,E2 -4076.729} C_VEL
LIN {X 0,Y 542.212,Z 150.61,A -85,B 0,C 180,E1 -4078.659,E2 -4078.659} C_VEL
LIN {X 0,Y 541.684,Z 147.437,A -85,B 0,C 180,E1 -4078.986,E2 -4078.986} C_VEL
LIN {X 0,Y 538.02,Z 135.095,A -85,B 0,C 180,E1 -4080.401,E2 -4080.401} C_VEL
LIN {X 0,Y 538.049,Z 135.09,A -85,B 0,C 180,E1 -4083.283,E2 -4083.283} C_VEL
LIN {X 0,Y 537.991,Z 135.099,A -85,B 0,C 180,E1 -4086.006,E2 -4086.006} C_VEL
LIN {X 0,Y 538.009,Z 135.092,A -85,B 0,C 180,E1 -4088.832,E2 -4088.832} C_VEL
LIN {X 0,Y 537.981,Z 135.098,A -85,B 0,C 180,E1 -4091.873,E2 -4091.873} C_VEL
LIN {X 0,Y 537.991,Z 135.095,A -85,B 0,C 180,E1 -4094.865,E2 -4094.865} C_VEL
LIN {X 0,Y 537.972,Z 135.102,A -85,B 0,C 180,E1 -4097.209,E2 -4097.209} C_VEL
LIN {X 0,Y 537.978,Z 135.095,A -85,B 0,C 180,E1 -4100.423,E2 -4100.423} C_VEL
LIN {X 0,Y 537.956,Z 135.104,A -85,B 0,C 180,E1 -4103.062,E2 -4103.062} C_VEL
LIN {X 0,Y 537.998,Z 135.093,A -85,B 0,C 180,E1 -4105.825,E2 -4105.825} C_VEL
LIN {X 0,Y 537.992,Z 135.098,A -85,B 0,C 180,E1 -4108.498,E2 -4108.498} C_VEL
LIN {X 0,Y 538.005,Z 135.096,A -85,B 0,C 180,E1 -4111.097,E2 -4111.097} C_VEL
LIN {X 0,Y 537.994,Z 135.098,A -85,B 0,C 180,E1 -4113.631,E2 -4113.631} C_VEL
LIN {X 0,Y 538.023,Z 135.154,A -85,B 0,C 180,E1 -4115.06,E2 -4115.06} C_VEL
LIN {X 0,Y 540.329,Z 145.023,A -85,B 0,C 180,E1 -4116.83,E2 -4116.83} C_VEL
LIN {X 0,Y 540.067,Z 157.529,A -85,B 0,C 180,E1 -4118.831,E2 -4118.831} C_VEL
LIN {X 0,Y 539.478,Z 176.248,A -85,B 0,C 180,E1 -4121.781,E2 -4121.781} C_VEL
LIN {X 0,Y 538.998,Z 193.951,A -85,B 0,C 180,E1 -4124.535,E2 -4124.535} C_VEL
LIN {X 0,Y 538.917,Z 197.577,A -85,B 0,C 180,E1 -4125.096,E2 -4125.096} C_VEL
LIN {X 0,Y 540.151,Z 203.231,A -85,B 0,C 180,E1 -4125.233,E2 -4125.233} C_VEL
LIN {X 0,Y 539.411,Z 308.278,A -85,B 0,C 180,E1 -4126.82,E2 -4126.82} C_VEL
LIN {X 0,Y 539.283,Z 322.229,A -85,B 0,C 180,E1 -4127.2,E2 -4127.2} C_VEL
LIN {X 0,Y 539.167,Z 334.298,A -85,B 0,C 180,E1 -4127.685,E2 -4127.685} C_VEL
LIN {X 0,Y 538.927,Z 346.698,A -85,B 0,C 180,E1 -4128.353,E2 -4128.353} C_VEL
LIN {X 0,Y 538.731,Z 357.503,A -85,B 0,C 180,E1 -4129.096,E2 -4129.096} C_VEL
LIN {X 0,Y 538.512,Z 366.436,A -85,B 0,C 180,E1 -4129.852,E2 -4129.852} C_VEL
LIN {X 0,Y 538.325,Z 375.595,A -85,B 0,C 180,E1 -4130.797,E2 -4130.797} C_VEL
LIN {X 0,Y 538.121,Z 384.434,A -85,B 0,C 180,E1 -4131.929,E2 -4131.929} C_VEL
LIN {X 0,Y 537.948,Z 392.171,A -85,B 0,C 180,E1 -4133.171,E2 -4133.171} C_VEL
LIN {X 0,Y 537.851,Z 398.005,A -85,B 0,C 180,E1 -4134.376,E2 -4134.376} C_VEL
LIN {X 0,Y 537.782,Z 402.263,A -85,B 0,C 180,E1 -4135.503,E2 -4135.503} C_VEL
LIN {X 0,Y 537.727,Z 404.507,A -85,B 0,C 180,E1 -4136.253,E2 -4136.253} C_VEL
LIN {X 0,Y 537.689,Z 406.33,A -85,B 0,C 180,E1 -4137.003,E2 -4137.003} C_VEL
LIN {X 0,Y 537.644,Z 407.712,A -85,B 0,C 180,E1 -4137.753,E2 -4137.753} C_VEL
LIN {X 0,Y 537.625,Z 409.269,A -85,B 0,C 180,E1 -4139.251,E2 -4139.251} C_VEL
LIN {X 0,Y 537.617,Z 409.479,A -85,B 0,C 180,E1 -4140,E2 -4140} C_VEL
LIN {X 0,Y 537.624,Z 409.28,A -85,B 0,C 180,E1 -4140.749,E2 -4140.749} C_VEL
LIN {X 0,Y 537.643,Z 407.716,A -85,B 0,C 180,E1 -4142.248,E2 -4142.248} C_VEL
LIN {X 0,Y 537.667,Z 406.345,A -85,B 0,C 180,E1 -4142.997,E2 -4142.997} C_VEL
LIN {X 0,Y 537.753,Z 403.469,A -85,B 0,C 180,E1 -4144.122,E2 -4144.122} C_VEL
LIN {X 0,Y 537.696,Z 399.601,A -85,B 0,C 180,E1 -4145.25,E2 -4145.25} C_VEL
LIN {X 0,Y 537.87,Z 394.244,A -85,B 0,C 180,E1 -4146.445,E2 -4146.445} C_VEL
LIN {X 0,Y 537.973,Z 387.066,A -85,B 0,C 180,E1 -4147.695,E2 -4147.695} C_VEL
LIN {X 0,Y 538.15,Z 378.889,A -85,B 0,C 180,E1 -4148.827,E2 -4148.827} C_VEL
LIN {X 0,Y 538.348,Z 370.509,A -85,B 0,C 180,E1 -4149.771,E2 -4149.771} C_VEL
LIN {X 0,Y 538.597,Z 360.151,A -85,B 0,C 180,E1 -4150.716,E2 -4150.716} C_VEL
LIN {X 0,Y 538.793,Z 348.653,A -85,B 0,C 180,E1 -4151.556,E2 -4151.556} C_VEL
LIN {X 0,Y 539.023,Z 336.778,A -85,B 0,C 180,E1 -4152.232,E2 -4152.232} C_VEL
LIN {X 0,Y 539.088,Z 324.659,A -85,B 0,C 180,E1 -4152.757,E2 -4152.757} C_VEL
LIN {X 0,Y 539.305,Z 311.49,A -85,B 0,C 180,E1 -4153.159,E2 -4153.159} C_VEL
